LIN {X 0,Y 129.168,Z 1032.646,A -85,B 0,C 180,E1 7073.413,E2 7073.413} C_VEL
LIN {X 0,Y 137.523,Z 1024.267,A -85,B 0,C 180,E1 7063.963,E2 7063.963} C_VEL
LIN {X 0,Y 148.39,Z 1014.459,A -85,B 0,C 180,E1 7056.043,E2 7056.043} C_VEL
LIN {X 0,Y 160.932,Z 1003.211,A -85,B 0,C 180,E1 7049.563,E2 7049.563} C_VEL
LIN {X 0,Y 174.466,Z 990.679,A -85,B 0,C 180,E1 7044.323,E2 7044.323} C_VEL
LIN {X 0,Y 188.456,Z 977.034,A -85,B 0,C 180,E1 7040.101,E2 7040.101} C_VEL
LIN {X 0,Y 202.822,Z 961.714,A -85,B 0,C 180,E1 7036.613,E2 7036.613} C_VEL
LIN {X 0,Y 217.2,Z 944.88,A -85,B 0,C 180,E1 7033.754,E2 7033.754} C_VEL
LIN {X 0,Y 230.71,Z 927.31,A -85,B 0,C 180,E1 7031.498,E2 7031.498} C_VEL
LIN {X 0,Y 243.023,Z 909.185,A -85,B 0,C 180,E1 7029.742,E2 7029.742} C_VEL
LIN {X 0,Y 254.635,Z 889.694,A -85,B 0,C 180,E1 7028.302,E2 7028.302} C_VEL
LIN {X 0,Y 264.561,Z 870.602,A -85,B 0,C 180,E1 7027.217,E2 7027.217} C_VEL
LIN {X 0,Y 273.322,Z 850.557,A -85,B 0,C 180,E1 7026.358,E2 7026.358} C_VEL
LIN {X 0,Y 281.328,Z 828.424,A -85,B 0,C 180,E1 7025.647,E2 7025.647} C_VEL
LIN {X 0,Y 287.652,Z 806.092,A -85,B 0,C 180,E1 7025.074,E2 7025.074} C_VEL
LIN {X 0,Y 292.242,Z 783.432,A -85,B 0,C 180,E1 7024.59,E2 7024.59} C_VEL
LIN {X 0,Y 296.797,Z 747.071,A -85,B 0,C 180,E1 7023.93,E2 7023.93} C_VEL
LIN {X 0,Y 309.195,Z 637.344,A -85,B 0,C 180,E1 7021.992,E2 7021.992} C_VEL
LIN {X 0,Y 308.31,Z 635.045,A -85,B 0,C 180,E1 7019.999,E2 7019.999} C_VEL
LIN {X 0,Y 307.563,Z 632.464,A -85,B 0,C 180,E1 7017.018,E2 7017.018} C_VEL
LIN {X 0,Y 307.478,Z 632.463,A -85,B 0,C 180,E1 7012.663,E2 7012.663} C_VEL
LIN {X 0,Y 308.466,Z 636.029,A -85,B 0,C 180,E1 7008.785,E2 7008.785} C_VEL
LIN {X 0,Y 308.571,Z 636.609,A -85,B 0,C 180,E1 7008.484,E2 7008.484} C_VEL
LIN {X 0,Y 293.648,Z 770.192,A -85,B 0,C 180,E1 7006.284,E2 7006.284} C_VEL
LIN {X 0,Y 289.742,Z 791.809,A -85,B 0,C 180,E1 7005.734,E2 7005.734} C_VEL
LIN {X 0,Y 284.597,Z 812.246,A -85,B 0,C 180,E1 7005.05,E2 7005.05} C_VEL
LIN {X 0,Y 277.983,Z 832.312,A -85,B 0,C 180,E1 7004.188,E2 7004.188} C_VEL
LIN {X 0,Y 270.077,Z 851.641,A -85,B 0,C 180,E1 7003.139,E2 7003.139} C_VEL
LIN {X 0,Y 260.928,Z 870.394,A -85,B 0,C 180,E1 7001.866,E2 7001.866} C_VEL
LIN {X 0,Y 250.585,Z 888.261,A -85,B 0,C 180,E1 7000.334,E2 7000.334} C_VEL
LIN {X 0,Y 239.316,Z 905.023,A -85,B 0,C 180,E1 6998.52,E2 6998.52} C_VEL
LIN {X 0,Y 227.072,Z 920.973,A -85,B 0,C 180,E1 6996.332,E2 6996.332} C_VEL
LIN {X 0,Y 214.134,Z 935.705,A -85,B 0,C 180,E1 6993.704,E2 6993.704} C_VEL
LIN {X 0,Y 200.856,Z 949.005,A -85,B 0,C 180,E1 6990.593,E2 6990.593} C_VEL
LIN {X 0,Y 187.475,Z 961.017,A -85,B 0,C 180,E1 6986.86,E2 6986.86} C_VEL
LIN {X 0,Y 174.234,Z 971.657,A -85,B 0,C 180,E1 6982.367,E2 6982.367} C_VEL
LIN {X 0,Y 161.499,Z 980.804,A -85,B 0,C 180,E1 6976.933,E2 6976.933} C_VEL
LIN {X 0,Y 149.251,Z 988.867,A -85,B 0,C 180,E1 6970.025,E2 6970.025} C_VEL
LIN {X 0,Y 139.655,Z 994.788,A -85,B 0,C 180,E1 6962.477,E2 6962.477} C_VEL
LIN {X 0,Y 132.062,Z 999.229,A -85,B 0,C 180,E1 6953.634,E2 6953.634} C_VEL
LIN {X 0,Y 127.304,Z 1001.968,A -85,B 0,C 180,E1 6944.092,E2 6944.092} C_VEL
LIN {X 0,Y 125.173,Z 1003.266,A -85,B 0,C 180,E1 6934.123,E2 6934.123} C_VEL
LIN {X 0,Y 125.206,Z 1003.258,A -85,B 0,C 180,E1 6925.42,E2 6925.42} C_VEL
LIN {X 0,Y 127.437,Z 1001.916,A -85,B 0,C 180,E1 6915.459,E2 6915.459} C_VEL
LIN {X 0,Y 132.311,Z 999.12,A -85,B 0,C 180,E1 6905.916,E2 6905.916} C_VEL
LIN {X 0,Y 140,Z 994.662,A -85,B 0,C 180,E1 6897.127,E2 6897.127} C_VEL
LIN {X 0,Y 149.777,Z 988.636,A -85,B 0,C 180,E1 6889.556,E2 6889.556} C_VEL
LIN {X 0,Y 162.013,Z 980.566,A -85,B 0,C 180,E1 6882.743,E2 6882.743} C_VEL
LIN {X 0,Y 174.948,Z 971.227,A -85,B 0,C 180,E1 6877.288,E2 6877.288} C_VEL
LIN {X 0,Y 188.83,Z 960.069,A -85,B 0,C 180,E1 6872.657,E2 6872.657} C_VEL
LIN {X 0,Y 202.291,Z 947.848,A -85,B 0,C 180,E1 6868.971,E2 6868.971} C_VEL
LIN {X 0,Y 216.428,Z 933.414,A -85,B 0,C 180,E1 6865.727,E2 6865.727} C_VEL
LIN {X 0,Y 229.449,Z 918.328,A -85,B 0,C 180,E1 6863.151,E2 6863.151} C_VEL
LIN {X 0,Y 241.141,Z 902.814,A -85,B 0,C 180,E1 6861.102,E2 6861.102} C_VEL
LIN {X 0,Y 252.636,Z 885.258,A -85,B 0,C 180,E1 6859.279,E2 6859.279} C_VEL
LIN {X 0,Y 263.01,Z 866.832,A -85,B 0,C 180,E1 6857.767,E2 6857.767} C_VEL
LIN {X 0,Y 272.187,Z 847.478,A -85,B 0,C 180,E1 6856.51,E2 6856.51} C_VEL
LIN {X 0,Y 279.844,Z 827.707,A -85,B 0,C 180,E1 6855.495,E2 6855.495} C_VEL
LIN {X 0,Y 286.583,Z 805.859,A -85,B 0,C 180,E1 6854.618,E2 6854.618} C_VEL
LIN {X 0,Y 291.486,Z 784.725,A -85,B 0,C 180,E1 6853.967,E2 6853.967} C_VEL
LIN {X 0,Y 294.809,Z 763.059,A -85,B 0,C 180,E1 6853.473,E2 6853.473} C_VEL
LIN {X 0,Y 308.856,Z 636.573,A -85,B 0,C 180,E1 6851.39,E2 6851.39} C_VEL
LIN {X 0,Y 308.132,Z 634.469,A -85,B 0,C 180,E1 6849.338,E2 6849.338} C_VEL
LIN {X 0,Y 307.66,Z 632.494,A -85,B 0,C 180,E1 6846.719,E2 6846.719} C_VEL
LIN {X 0,Y 307.835,Z 632.739,A -85,B 0,C 180,E1 6842.793,E2 6842.793} C_VEL
LIN {X 0,Y 309.082,Z 636.612,A -85,B 0,C 180,E1 6838.703,E2 6838.703} C_VEL
LIN {X 0,Y 309.408,Z 637.777,A -85,B 0,C 180,E1 6837.963,E2 6837.963} C_VEL
LIN {X 0,Y 296.291,Z 753.366,A -85,B 0,C 180,E1 6835.967,E2 6835.967} C_VEL
LIN {X 0,Y 295.27,Z 761.06,A -85,B 0,C 180,E1 6836.032,E2 6836.032} C_VEL
LIN {X 0,Y 291.656,Z 781.543,A -85,B 0,C 180,E1 6836.883,E2 6836.883} C_VEL
LIN {X 0,Y 290.371,Z 788.084,A -85,B 0,C 180,E1 6836.883,E2 6836.883} C_VEL
LIN {X 0,Y 284.988,Z 811.855,A -85,B 0,C 180,E1 6836.38,E2 6836.38} C_VEL
LIN {X 0,Y 278.446,Z 833.355,A -85,B 0,C 180,E1 6835.84,E2 6835.84} C_VEL
LIN {X 0,Y 269.935,Z 855.2,A -85,B 0,C 180,E1 6835.14,E2 6835.14} C_VEL
LIN {X 0,Y 260.279,Z 875.739,A -85,B 0,C 180,E1 6834.24,E2 6834.24} C_VEL
LIN {X 0,Y 249.372,Z 895.581,A -85,B 0,C 180,E1 6833.092,E2 6833.092} C_VEL
LIN {X 0,Y 237.943,Z 913.511,A -85,B 0,C 180,E1 6831.73,E2 6831.73} C_VEL
LIN {X 0,Y 224.47,Z 932.114,A -85,B 0,C 180,E1 6829.87,E2 6829.87} C_VEL
LIN {X 0,Y 210.848,Z 948.889,A -85,B 0,C 180,E1 6827.654,E2 6827.654} C_VEL
LIN {X 0,Y 196.469,Z 964.671,A -85,B 0,C 180,E1 6824.862,E2 6824.862} C_VEL
LIN {X 0,Y 181.547,Z 979.576,A -85,B 0,C 180,E1 6821.314,E2 6821.314} C_VEL
LIN {X 0,Y 166.472,Z 993.481,A -85,B 0,C 180,E1 6816.773,E2 6816.773} C_VEL
LIN {X 0,Y 151.986,Z 1005.938,A -85,B 0,C 180,E1 6811.04,E2 6811.04} C_VEL
LIN {X 0,Y 138.719,Z 1016.968,A -85,B 0,C 180,E1 6803.831,E2 6803.831} C_VEL
LIN {X 0,Y 127.52,Z 1026.514,A -85,B 0,C 180,E1 6794.884,E2 6794.884} C_VEL
LIN {X 0,Y 119.945,Z 1033.8,A -85,B 0,C 180,E1 6785.113,E2 6785.113} C_VEL
LIN {X 0,Y 115.716,Z 1039.287,A -85,B 0,C 180,E1 6774.504,E2 6774.504} C_VEL
LIN {X 0,Y 114.694,Z 1042.845,A -85,B 0,C 180,E1 6764.619,E2 6764.619} C_VEL
LIN {X 0,Y 115.455,Z 1044.705,A -85,B 0,C 180,E1 6755.965,E2 6755.965} C_VEL
LIN {X 0,Y 116.042,Z 1045.172,A -85,B 0,C 180,E1 6750.494,E2 6750.494} C_VEL
LIN {X 0,Y 115.673,Z 1044.857,A -85,B 0,C 180,E1 6745.538,E2 6745.538} C_VEL
LIN {X 0,Y 114.765,Z 1043.356,A -85,B 0,C 180,E1 6737.354,E2 6737.354} C_VEL
LIN {X 0,Y 115.389,Z 1039.917,A -85,B 0,C 180,E1 6727.05,E2 6727.05} C_VEL
LIN {X 0,Y 118.623,Z 1035.213,A -85,B 0,C 180,E1 6717.354,E2 6717.354} C_VEL
LIN {X 0,Y 125.827,Z 1027.96,A -85,B 0,C 180,E1 6706.891,E2 6706.891} C_VEL
LIN {X 0,Y 135.903,Z 1019.293,A -85,B 0,C 180,E1 6698.073,E2 6698.073} C_VEL
LIN {X 0,Y 147.961,Z 1009.202,A -85,B 0,C 180,E1 6690.882,E2 6690.882} C_VEL
LIN {X 0,Y 162.033,Z 997.214,A -85,B 0,C 180,E1 6684.809,E2 6684.809} C_VEL
LIN {X 0,Y 176.659,Z 984.102,A -85,B 0,C 180,E1 6680.026,E2 6680.026} C_VEL
LIN {X 0,Y 191.59,Z 969.538,A -85,B 0,C 180,E1 6676.207,E2 6676.207} C_VEL
LIN {X 0,Y 206.378,Z 953.698,A -85,B 0,C 180,E1 6673.142,E2 6673.142} C_VEL
LIN {X 0,Y 220.798,Z 936.614,A -85,B 0,C 180,E1 6670.683,E2 6670.683} C_VEL
LIN {X 0,Y 233.725,Z 919.31,A -85,B 0,C 180,E1 6668.807,E2 6668.807} C_VEL
LIN {X 0,Y 245.951,Z 900.785,A -85,B 0,C 180,E1 6667.282,E2 6667.282} C_VEL
LIN {X 0,Y 256.915,Z 881.888,A -85,B 0,C 180,E1 6666.087,E2 6666.087} C_VEL
LIN {X 0,Y 267.025,Z 861.28,A -85,B 0,C 180,E1 6665.106,E2 6665.106} C_VEL
LIN {X 0,Y 276.006,Z 839.357,A -85,B 0,C 180,E1 6664.342,E2 6664.342} C_VEL
LIN {X 0,Y 283.32,Z 817.128,A -85,B 0,C 180,E1 6663.751,E2 6663.751} C_VEL
LIN {X 0,Y 288.927,Z 794.538,A -85,B 0,C 180,E1 6663.252,E2 6663.252} C_VEL
LIN {X 0,Y 292.707,Z 771.832,A -85,B 0,C 180,E1 6662.822,E2 6662.822} C_VEL
LIN {X 0,Y 307.568,Z 643.681,A -85,B 0,C 180,E1 6660.651,E2 6660.651} C_VEL
LIN {X 0,Y 306.554,Z 640.371,A -85,B 0,C 180,E1 6656.821,E2 6656.821} C_VEL
LIN {X 0,Y 306.492,Z 640.482,A -85,B 0,C 180,E1 6652.69,E2 6652.69} C_VEL
LIN {X 0,Y 307.068,Z 643.011,A -85,B 0,C 180,E1 6649.87,E2 6649.87} C_VEL
LIN {X 0,Y 292.446,Z 770.849,A -85,B 0,C 180,E1 6647.825,E2 6647.825} C_VEL
LIN {X 0,Y 288.464,Z 792.458,A -85,B 0,C 180,E1 6647.294,E2 6647.294} C_VEL
LIN {X 0,Y 283.142,Z 813.196,A -85,B 0,C 180,E1 6646.626,E2 6646.626} C_VEL
LIN {X 0,Y 276.411,Z 833.238,A -85,B 0,C 180,E1 6645.799,E2 6645.799} C_VEL
LIN {X 0,Y 268.363,Z 852.557,A -85,B 0,C 180,E1 6644.793,E2 6644.793} C_VEL
LIN {X 0,Y 259.043,Z 871.321,A -85,B 0,C 180,E1 6643.572,E2 6643.572} C_VEL
LIN {X 0,Y 248.495,Z 889.202,A -85,B 0,C 180,E1 6642.102,E2 6642.102} C_VEL
LIN {X 0,Y 236.791,Z 906.255,A -85,B 0,C 180,E1 6640.328,E2 6640.328} C_VEL
LIN {X 0,Y 224.876,Z 921.49,A -85,B 0,C 180,E1 6638.323,E2 6638.323} C_VEL
LIN {X 0,Y 211.579,Z 936.29,A -85,B 0,C 180,E1 6635.792,E2 6635.792} C_VEL
LIN {X 0,Y 197.89,Z 949.707,A -85,B 0,C 180,E1 6632.781,E2 6632.781} C_VEL
LIN {X 0,Y 184.024,Z 961.824,A -85,B 0,C 180,E1 6629.145,E2 6629.145} C_VEL
LIN {X 0,Y 170.215,Z 972.521,A -85,B 0,C 180,E1 6624.736,E2 6624.736} C_VEL
LIN {X 0,Y 156.826,Z 981.768,A -85,B 0,C 180,E1 6619.35,E2 6619.35} C_VEL
LIN {X 0,Y 144.365,Z 989.606,A -85,B 0,C 180,E1 6612.746,E2 6612.746} C_VEL
LIN {X 0,Y 133.912,Z 995.704,A -85,B 0,C 180,E1 6605.095,E2 6605.095} C_VEL
LIN {X 0,Y 125.479,Z 1000.232,A -85,B 0,C 180,E1 6595.993,E2 6595.993} C_VEL
LIN {X 0,Y 120.003,Z 1003.146,A -85,B 0,C 180,E1 6585.959,E2 6585.959} C_VEL
LIN {X 0,Y 117.473,Z 1004.583,A -85,B 0,C 180,E1 6575.862,E2 6575.862} C_VEL
LIN {X 0,Y 117.248,Z 1004.661,A -85,B 0,C 180,E1 6566.174,E2 6566.174} C_VEL
LIN {X 0,Y 119.465,Z 1003.476,A -85,B 0,C 180,E1 6555.458,E2 6555.458} C_VEL
LIN {X 0,Y 124.517,Z 1000.849,A -85,B 0,C 180,E1 6545.319,E2 6545.319} C_VEL
LIN {X 0,Y 132.538,Z 996.484,A -85,B 0,C 180,E1 6536.065,E2 6536.065} C_VEL
LIN {X 0,Y 143.196,Z 990.387,A -85,B 0,C 180,E1 6527.908,E2 6527.908} C_VEL
LIN {X 0,Y 156.111,Z 982.368,A -85,B 0,C 180,E1 6520.907,E2 6520.907} C_VEL
LIN {X 0,Y 169.428,Z 973.26,A -85,B 0,C 180,E1 6515.472,E2 6515.472} C_VEL
LIN {X 0,Y 183.179,Z 962.654,A -85,B 0,C 180,E1 6511.022,E2 6511.022} C_VEL
LIN {X 0,Y 197.009,Z 950.72,A -85,B 0,C 180,E1 6507.356,E2 6507.356} C_VEL
LIN {X 0,Y 210.672,Z 937.502,A -85,B 0,C 180,E1 6504.322,E2 6504.322} C_VEL
LIN {X 0,Y 224.136,Z 922.594,A -85,B 0,C 180,E1 6501.732,E2 6501.732} C_VEL
LIN {X 0,Y 236.704,Z 906.685,A -85,B 0,C 180,E1 6499.613,E2 6499.613} C_VEL
LIN {X 0,Y 248.412,Z 889.718,A -85,B 0,C 180,E1 6497.839,E2 6497.839} C_VEL
LIN {X 0,Y 258.896,Z 871.998,A -85,B 0,C 180,E1 6496.376,E2 6496.376} C_VEL
LIN {X 0,Y 268.285,Z 853.243,A -85,B 0,C 180,E1 6495.146,E2 6495.146} C_VEL
LIN {X 0,Y 276.339,Z 834.11,A -85,B 0,C 180,E1 6494.142,E2 6494.142} C_VEL
LIN {X 0,Y 283.07,Z 814.201,A -85,B 0,C 180,E1 6493.313,E2 6493.313} C_VEL
LIN {X 0,Y 288.641,Z 792.794,A -85,B 0,C 180,E1 6492.619,E2 6492.619} C_VEL
LIN {X 0,Y 292.691,Z 770.866,A -85,B 0,C 180,E1 6492.078,E2 6492.078} C_VEL
LIN {X 0,Y 307.388,Z 643.047,A -85,B 0,C 180,E1 6490.032,E2 6490.032} C_VEL
LIN {X 0,Y 306.668,Z 640.418,A -85,B 0,C 180,E1 6486.553,E2 6486.553} C_VEL
LIN {X 0,Y 306.827,Z 640.61,A -85,B 0,C 180,E1 6482.989,E2 6482.989} C_VEL
LIN {X 0,Y 307.792,Z 643.979,A -85,B 0,C 180,E1 6479.341,E2 6479.341} C_VEL
LIN {X 0,Y 291.953,Z 779.066,A -85,B 0,C 180,E1 6477.056,E2 6477.056} C_VEL
LIN {X 0,Y 290.371,Z 788.084,A -85,B 0,C 180,E1 6476.883,E2 6476.883} C_VEL
LIN {X 0,Y 288.487,Z 796.75,A -85,B 0,C 180,E1 6476.959,E2 6476.959} C_VEL
LIN {X 0,Y 283.247,Z 814.649,A -85,B 0,C 180,E1 6477.719,E2 6477.719} C_VEL
LIN {X 0,Y 280.857,Z 822.038,A -85,B 0,C 180,E1 6477.749,E2 6477.749} C_VEL
LIN {X 0,Y 273.293,Z 843.641,A -85,B 0,C 180,E1 6477.187,E2 6477.187} C_VEL
LIN {X 0,Y 264.46,Z 863.924,A -85,B 0,C 180,E1 6476.495,E2 6476.495} C_VEL
LIN {X 0,Y 253.739,Z 884.733,A -85,B 0,C 180,E1 6475.528,E2 6475.528} C_VEL
LIN {X 0,Y 241.855,Z 904.472,A -85,B 0,C 180,E1 6474.307,E2 6474.307} C_VEL
LIN {X 0,Y 228.794,Z 923.101,A -85,B 0,C 180,E1 6472.76,E2 6472.76} C_VEL
LIN {X 0,Y 214.271,Z 941.356,A -85,B 0,C 180,E1 6470.729,E2 6470.729} C_VEL
LIN {X 0,Y 199.18,Z 958.205,A -85,B 0,C 180,E1 6468.204,E2 6468.204} C_VEL
LIN {X 0,Y 184.148,Z 973.242,A -85,B 0,C 180,E1 6465.125,E2 6465.125} C_VEL
LIN {X 0,Y 168.946,Z 987.038,A -85,B 0,C 180,E1 6461.249,E2 6461.249} C_VEL
LIN {X 0,Y 153.586,Z 999.968,A -85,B 0,C 180,E1 6456.196,E2 6456.196} C_VEL
LIN {X 0,Y 138.967,Z 1011.527,A -85,B 0,C 180,E1 6449.701,E2 6449.701} C_VEL
LIN {X 0,Y 126.225,Z 1021.348,A -85,B 0,C 180,E1 6441.647,E2 6441.647} C_VEL
LIN {X 0,Y 115.942,Z 1029.738,A -85,B 0,C 180,E1 6431.608,E2 6431.608} C_VEL
LIN {X 0,Y 109.765,Z 1035.768,A -85,B 0,C 180,E1 6421.105,E2 6421.105} C_VEL
LIN {X 0,Y 106.923,Z 1040.415,A -85,B 0,C 180,E1 6409.105,E2 6409.105} C_VEL
LIN {X 0,Y 107.097,Z 1042.759,A -85,B 0,C 180,E1 6399.674,E2 6399.674} C_VEL
LIN {X 0,Y 108.056,Z 1043.707,A -85,B 0,C 180,E1 6392.121,E2 6392.121} C_VEL
LIN {X 0,Y 108.056,Z 1043.702,A -85,B 0,C 180,E1 6387.865,E2 6387.865} C_VEL
LIN {X 0,Y 107.097,Z 1042.746,A -85,B 0,C 180,E1 6380.325,E2 6380.325} C_VEL
LIN {X 0,Y 106.935,Z 1040.364,A -85,B 0,C 180,E1 6370.792,E2 6370.792} C_VEL
LIN {X 0,Y 109.83,Z 1035.655,A -85,B 0,C 180,E1 6358.74,E2 6358.74} C_VEL
LIN {X 0,Y 115.94,Z 1029.692,A -85,B 0,C 180,E1 6348.391,E2 6348.391} C_VEL
LIN {X 0,Y 125.683,Z 1021.706,A -85,B 0,C 180,E1 6338.772,E2 6338.772} C_VEL
LIN {X 0,Y 138.303,Z 1011.975,A -85,B 0,C 180,E1 6330.648,E2 6330.648} C_VEL
LIN {X 0,Y 152.423,Z 1000.778,A -85,B 0,C 180,E1 6324.242,E2 6324.242} C_VEL
LIN {X 0,Y 168.123,Z 987.622,A -85,B 0,C 180,E1 6318.984,E2 6318.984} C_VEL
LIN {X 0,Y 183.278,Z 973.924,A -85,B 0,C 180,E1 6315.068,E2 6315.068} C_VEL
LIN {X 0,Y 198.482,Z 958.727,A -85,B 0,C 180,E1 6311.919,E2 6311.919} C_VEL
LIN {X 0,Y 213.017,Z 942.589,A -85,B 0,C 180,E1 6309.455,E2 6309.455} C_VEL
LIN {X 0,Y 226.899,Z 925.402,A -85,B 0,C 180,E1 6307.476,E2 6307.476} C_VEL
LIN {X 0,Y 239.746,Z 907.253,A -85,B 0,C 180,E1 6305.917,E2 6305.917} C_VEL
LIN {X 0,Y 251.796,Z 887.736,A -85,B 0,C 180,E1 6304.651,E2 6304.651} C_VEL
LIN {X 0,Y 262.503,Z 867.622,A -85,B 0,C 180,E1 6303.668,E2 6303.668} C_VEL
LIN {X 0,Y 271.325,Z 847.873,A -85,B 0,C 180,E1 6302.955,E2 6302.955} C_VEL
LIN {X 0,Y 279.201,Z 826.422,A -85,B 0,C 180,E1 6302.366,E2 6302.366} C_VEL
LIN {X 0,Y 285.552,Z 804.428,A -85,B 0,C 180,E1 6301.871,E2 6301.871} C_VEL
LIN {X 0,Y 290.209,Z 781.99,A -85,B 0,C 180,E1 6301.439,E2 6301.439} C_VEL
LIN {X 0,Y 294.604,Z 748.025,A -85,B 0,C 180,E1 6300.864,E2 6300.864} C_VEL
LIN {X 0,Y 306.041,Z 650.45,A -85,B 0,C 180,E1 6299.251,E2 6299.251} C_VEL
LIN {X 0,Y 305.538,Z 648.282,A -85,B 0,C 180,E1 6296.623,E2 6296.623} C_VEL
LIN {X 0,Y 305.497,Z 648.381,A -85,B 0,C 180,E1 6292.855,E2 6292.855} C_VEL
LIN {X 0,Y 305.695,Z 649.877,A -85,B 0,C 180,E1 6291.262,E2 6291.262} C_VEL
LIN {X 0,Y 291.442,Z 771.609,A -85,B 0,C 180,E1 6289.376,E2 6289.376} C_VEL
LIN {X 0,Y 287.374,Z 793.238,A -85,B 0,C 180,E1 6288.864,E2 6288.864} C_VEL
LIN {X 0,Y 281.903,Z 814.147,A -85,B 0,C 180,E1 6288.217,E2 6288.217} C_VEL
LIN {X 0,Y 275.157,Z 833.898,A -85,B 0,C 180,E1 6287.439,E2 6287.439} C_VEL
LIN {X 0,Y 266.876,Z 853.472,A -85,B 0,C 180,E1 6286.466,E2 6286.466} C_VEL
LIN {X 0,Y 257.391,Z 872.246,A -85,B 0,C 180,E1 6285.301,E2 6285.301} C_VEL
LIN {X 0,Y 246.645,Z 890.141,A -85,B 0,C 180,E1 6283.897,E2 6283.897} C_VEL
LIN {X 0,Y 234.705,Z 907.222,A -85,B 0,C 180,E1 6282.201,E2 6282.201} C_VEL
LIN {X 0,Y 222.091,Z 922.974,A -85,B 0,C 180,E1 6280.208,E2 6280.208} C_VEL
LIN {X 0,Y 208.474,Z 937.753,A -85,B 0,C 180,E1 6277.767,E2 6277.767} C_VEL
LIN {X 0,Y 194.408,Z 951.135,A -85,B 0,C 180,E1 6274.849,E2 6274.849} C_VEL
LIN {X 0,Y 180.098,Z 963.223,A -85,B 0,C 180,E1 6271.305,E2 6271.305} C_VEL
LIN {X 0,Y 165.774,Z 973.918,A -85,B 0,C 180,E1 6266.97,E2 6266.97} C_VEL
LIN {X 0,Y 151.784,Z 983.155,A -85,B 0,C 180,E1 6261.62,E2 6261.62} C_VEL
LIN {X 0,Y 138.065,Z 991.298,A -85,B 0,C 180,E1 6254.626,E2 6254.626} C_VEL
LIN {X 0,Y 127.029,Z 997.31,A -85,B 0,C 180,E1 6246.742,E2 6246.742} C_VEL
LIN {X 0,Y 118.069,Z 1001.787,A -85,B 0,C 180,E1 6237.213,E2 6237.213} C_VEL
LIN {X 0,Y 112.224,Z 1004.609,A -85,B 0,C 180,E1 6226.565,E2 6226.565} C_VEL
LIN {X 0,Y 109.562,Z 1005.964,A -85,B 0,C 180,E1 6215.762,E2 6215.762} C_VEL
LIN {X 0,Y 109.388,Z 1006.024,A -85,B 0,C 180,E1 6205.807,E2 6205.807} C_VEL
LIN {X 0,Y 111.832,Z 1004.845,A -85,B 0,C 180,E1 6194.441,E2 6194.441} C_VEL
LIN {X 0,Y 117.364,Z 1002.22,A -85,B 0,C 180,E1 6183.704,E2 6183.704} C_VEL
LIN {X 0,Y 126.156,Z 997.795,A -85,B 0,C 180,E1 6173.943,E2 6173.943} C_VEL
LIN {X 0,Y 137.413,Z 991.761,A -85,B 0,C 180,E1 6165.691,E2 6165.691} C_VEL
LIN {X 0,Y 150.381,Z 984.171,A -85,B 0,C 180,E1 6158.929,E2 6158.929} C_VEL
LIN {X 0,Y 164.233,Z 975.143,A -85,B 0,C 180,E1 6153.481,E2 6153.481} C_VEL
LIN {X 0,Y 178.458,Z 964.644,A -85,B 0,C 180,E1 6149.069,E2 6149.069} C_VEL
LIN {X 0,Y 193.509,Z 952.138,A -85,B 0,C 180,E1 6145.28,E2 6145.28} C_VEL
LIN {X 0,Y 207.552,Z 938.958,A -85,B 0,C 180,E1 6142.34,E2 6142.34} C_VEL
LIN {X 0,Y 221.143,Z 924.293,A -85,B 0,C 180,E1 6139.874,E2 6139.874} C_VEL
LIN {X 0,Y 234.185,Z 908.224,A -85,B 0,C 180,E1 6137.804,E2 6137.804} C_VEL
LIN {X 0,Y 246.126,Z 891.355,A -85,B 0,C 180,E1 6136.103,E2 6136.103} C_VEL
LIN {X 0,Y 256.866,Z 873.582,A -85,B 0,C 180,E1 6134.692,E2 6134.692} C_VEL
LIN {X 0,Y 266.806,Z 854.148,A -85,B 0,C 180,E1 6133.471,E2 6133.471} C_VEL
LIN {X 0,Y 274.996,Z 835.02,A -85,B 0,C 180,E1 6132.513,E2 6132.513} C_VEL
LIN {X 0,Y 281.839,Z 815.133,A -85,B 0,C 180,E1 6131.721,E2 6131.721} C_VEL
LIN {X 0,Y 287.554,Z 793.588,A -85,B 0,C 180,E1 6131.05,E2 6131.05} C_VEL
LIN {X 0,Y 291.686,Z 771.686,A -85,B 0,C 180,E1 6130.53,E2 6130.53} C_VEL
LIN {X 0,Y 305.99,Z 649.959,A -85,B 0,C 180,E1 6128.645,E2 6128.645} C_VEL
LIN {X 0,Y 305.681,Z 648.342,A -85,B 0,C 180,E1 6126.386,E2 6126.386} C_VEL
LIN {X 0,Y 305.841,Z 648.653,A -85,B 0,C 180,E1 6122.999,E2 6122.999} C_VEL
LIN {X 0,Y 306.268,Z 650.919,A -85,B 0,C 180,E1 6120.721,E2 6120.721} C_VEL
LIN {X 0,Y 291.044,Z 778.478,A -85,B 0,C 180,E1 6118.631,E2 6118.631} C_VEL
LIN {X 0,Y 286.602,Z 800.907,A -85,B 0,C 180,E1 6118.206,E2 6118.206} C_VEL
LIN {X 0,Y 280.857,Z 822.038,A -85,B 0,C 180,E1 6117.749,E2 6117.749} C_VEL
LIN {X 0,Y 278.71,Z 828.32,A -85,B 0,C 180,E1 6117.788,E2 6117.788} C_VEL
LIN {X 0,Y 271.025,Z 846.672,A -85,B 0,C 180,E1 6118.528,E2 6118.528} C_VEL
LIN {X 0,Y 267.887,Z 853.694,A -85,B 0,C 180,E1 6118.555,E2 6118.555} C_VEL
LIN {X 0,Y 267.456,Z 854.699,A -85,B 0,C 180,E1 6118.529,E2 6118.529} C_VEL
LIN {X 0,Y 257.707,Z 874.676,A -85,B 0,C 180,E1 6117.777,E2 6117.777} C_VEL
LIN {X 0,Y 246.356,Z 894.548,A -85,B 0,C 180,E1 6116.779,E2 6116.779} C_VEL
LIN {X 0,Y 234.221,Z 912.856,A -85,B 0,C 180,E1 6115.562,E2 6115.562} C_VEL
LIN {X 0,Y 221.038,Z 930.208,A -85,B 0,C 180,E1 6114.029,E2 6114.029} C_VEL
LIN {X 0,Y 206.003,Z 947.754,A -85,B 0,C 180,E1 6111.949,E2 6111.949} C_VEL
LIN {X 0,Y 190.924,Z 963.362,A -85,B 0,C 180,E1 6109.439,E2 6109.439} C_VEL
LIN {X 0,Y 174.687,Z 978.393,A -85,B 0,C 180,E1 6106.091,E2 6106.091} C_VEL
LIN {X 0,Y 157.987,Z 992.406,A -85,B 0,C 180,E1 6101.681,E2 6101.681} C_VEL
LIN {X 0,Y 142.161,Z 1004.676,A -85,B 0,C 180,E1 6096.112,E2 6096.112} C_VEL
LIN {X 0,Y 127.337,Z 1015.413,A -85,B 0,C 180,E1 6088.857,E2 6088.857} C_VEL
LIN {X 0,Y 114.46,Z 1024.672,A -85,B 0,C 180,E1 6079.463,E2 6079.463} C_VEL
LIN {X 0,Y 105.447,Z 1031.771,A -85,B 0,C 180,E1 6068.743,E2 6068.743} C_VEL
LIN {X 0,Y 100.221,Z 1037.052,A -85,B 0,C 180,E1 6056.676,E2 6056.676} C_VEL
LIN {X 0,Y 98.852,Z 1040.548,A -85,B 0,C 180,E1 6044.647,E2 6044.647} C_VEL
LIN {X 0,Y 99.737,Z 1042.092,A -85,B 0,C 180,E1 6035.176,E2 6035.176} C_VEL
LIN {X 0,Y 100.286,Z 1042.459,A -85,B 0,C 180,E1 6030,E2 6030} C_VEL
LIN {X 0,Y 99.649,Z 1042.032,A -85,B 0,C 180,E1 6024.241,E2 6024.241} C_VEL
LIN {X 0,Y 98.845,Z 1040.293,A -85,B 0,C 180,E1 6014.15,E2 6014.15} C_VEL
LIN {X 0,Y 100.557,Z 1036.581,A -85,B 0,C 180,E1 6002.138,E2 6002.138} C_VEL
LIN {X 0,Y 106.149,Z 1031.133,A -85,B 0,C 180,E1 5990.169,E2 5990.169} C_VEL
LIN {X 0,Y 115.494,Z 1023.865,A -85,B 0,C 180,E1 5979.601,E2 5979.601} C_VEL
LIN {X 0,Y 128.651,Z 1014.37,A -85,B 0,C 180,E1 5970.381,E2 5970.381} C_VEL
LIN {X 0,Y 143.239,Z 1003.742,A -85,B 0,C 180,E1 5963.444,E2 5963.444} C_VEL
LIN {X 0,Y 158.811,Z 991.641,A -85,B 0,C 180,E1 5958.068,E2 5958.068} C_VEL
LIN {X 0,Y 175.044,Z 977.914,A -85,B 0,C 180,E1 5953.819,E2 5953.819} C_VEL
LIN {X 0,Y 191.18,Z 962.907,A -85,B 0,C 180,E1 5950.506,E2 5950.506} C_VEL
LIN {X 0,Y 206.469,Z 947.04,A -85,B 0,C 180,E1 5947.973,E2 5947.973} C_VEL
LIN {X 0,Y 221.161,Z 929.783,A -85,B 0,C 180,E1 5945.946,E2 5945.946} C_VEL
LIN {X 0,Y 235.139,Z 911.188,A -85,B 0,C 180,E1 5944.328,E2 5944.328} C_VEL
LIN {X 0,Y 247.334,Z 892.642,A -85,B 0,C 180,E1 5943.12,E2 5943.12} C_VEL
LIN {X 0,Y 258.152,Z 873.387,A -85,B 0,C 180,E1 5942.177,E2 5942.177} C_VEL
LIN {X 0,Y 268.047,Z 852.747,A -85,B 0,C 180,E1 5941.42,E2 5941.42} C_VEL
LIN {X 0,Y 276.543,Z 831.321,A -85,B 0,C 180,E1 5940.842,E2 5940.842} C_VEL
LIN {X 0,Y 283.406,Z 809.033,A -85,B 0,C 180,E1 5940.361,E2 5940.361} C_VEL
LIN {X 0,Y 288.65,Z 785.987,A -85,B 0,C 180,E1 5939.931,E2 5939.931} C_VEL
LIN {X 0,Y 292.268,Z 761.823,A -85,B 0,C 180,E1 5939.528,E2 5939.528} C_VEL
LIN {X 0,Y 304.702,Z 657.198,A -85,B 0,C 180,E1 5937.837,E2 5937.837} C_VEL
LIN {X 0,Y 304.518,Z 656.195,A -85,B 0,C 180,E1 5936.423,E2 5936.423} C_VEL
LIN {X 0,Y 304.505,Z 656.279,A -85,B 0,C 180,E1 5933.021,E2 5933.021} C_VEL
LIN {X 0,Y 304.509,Z 656.722,A -85,B 0,C 180,E1 5932.666,E2 5932.666} C_VEL
LIN {X 0,Y 290.654,Z 772.37,A -85,B 0,C 180,E1 5930.936,E2 5930.936} C_VEL
LIN {X 0,Y 286.501,Z 794.03,A -85,B 0,C 180,E1 5930.444,E2 5930.444} C_VEL
LIN {X 0,Y 280.884,Z 815.098,A -85,B 0,C 180,E1 5929.822,E2 5929.822} C_VEL
LIN {X 0,Y 273.934,Z 835.089,A -85,B 0,C 180,E1 5929.07,E2 5929.07} C_VEL
LIN {X 0,Y 265.619,Z 854.389,A -85,B 0,C 180,E1 5928.157,E2 5928.157} C_VEL
LIN {X 0,Y 255.977,Z 873.172,A -85,B 0,C 180,E1 5927.051,E2 5927.051} C_VEL
LIN {X 0,Y 245.042,Z 891.08,A -85,B 0,C 180,E1 5925.718,E2 5925.718} C_VEL
LIN {X 0,Y 232.874,Z 908.189,A -85,B 0,C 180,E1 5924.106,E2 5924.106} C_VEL
LIN {X 0,Y 219.553,Z 924.455,A -85,B 0,C 180,E1 5922.14,E2 5922.14} C_VEL
LIN {X 0,Y 205.624,Z 939.215,A -85,B 0,C 180,E1 5919.798,E2 5919.798} C_VEL
LIN {X 0,Y 191.188,Z 952.562,A -85,B 0,C 180,E1 5916.99,E2 5916.99} C_VEL
LIN {X 0,Y 175.637,Z 965.223,A -85,B 0,C 180,E1 5913.351,E2 5913.351} C_VEL
LIN {X 0,Y 160.842,Z 975.849,A -85,B 0,C 180,E1 5909.078,E2 5909.078} C_VEL
LIN {X 0,Y 146.3,Z 984.964,A -85,B 0,C 180,E1 5903.751,E2 5903.751} C_VEL
LIN {X 0,Y 132.54,Z 992.678,A -85,B 0,C 180,E1 5897.034,E2 5897.034} C_VEL
LIN {X 0,Y 120.765,Z 998.683,A -85,B 0,C 180,E1 5888.994,E2 5888.994} C_VEL
LIN {X 0,Y 111.083,Z 1003.161,A -85,B 0,C 180,E1 5879.082,E2 5879.082} C_VEL
LIN {X 0,Y 104.67,Z 1005.979,A -85,B 0,C 180,E1 5867.799,E2 5867.799} C_VEL
LIN {X 0,Y 101.718,Z 1007.33,A -85,B 0,C 180,E1 5856.208,E2 5856.208} C_VEL
LIN {X 0,Y 101.526,Z 1007.389,A -85,B 0,C 180,E1 5845.481,E2 5845.481} C_VEL
LIN {X 0,Y 104.236,Z 1006.215,A -85,B 0,C 180,E1 5833.276,E2 5833.276} C_VEL
LIN {X 0,Y 110.316,Z 1003.592,A -85,B 0,C 180,E1 5821.881,E2 5821.881} C_VEL
LIN {X 0,Y 119.703,Z 999.226,A -85,B 0,C 180,E1 5811.821,E2 5811.821} C_VEL
LIN {X 0,Y 131.855,Z 993.134,A -85,B 0,C 180,E1 5803.283,E2 5803.283} C_VEL
LIN {X 0,Y 145.531,Z 985.552,A -85,B 0,C 180,E1 5796.501,E2 5796.501} C_VEL
LIN {X 0,Y 160.759,Z 976.041,A -85,B 0,C 180,E1 5790.872,E2 5790.872} C_VEL
LIN {X 0,Y 175.553,Z 965.444,A -85,B 0,C 180,E1 5786.594,E2 5786.594} C_VEL
LIN {X 0,Y 191.107,Z 952.827,A -85,B 0,C 180,E1 5782.952,E2 5782.952} C_VEL
LIN {X 0,Y 205.545,Z 939.533,A -85,B 0,C 180,E1 5780.142,E2 5780.142} C_VEL
LIN {X 0,Y 219.83,Z 924.412,A -85,B 0,C 180,E1 5777.743,E2 5777.743} C_VEL
LIN {X 0,Y 232.8,Z 908.596,A -85,B 0,C 180,E1 5775.831,E2 5775.831} C_VEL
LIN {X 0,Y 244.973,Z 891.578,A -85,B 0,C 180,E1 5774.219,E2 5774.219} C_VEL
LIN {X 0,Y 255.911,Z 873.714,A -85,B 0,C 180,E1 5772.885,E2 5772.885} C_VEL
LIN {X 0,Y 265.557,Z 855.052,A -85,B 0,C 180,E1 5771.779,E2 5771.779} C_VEL
LIN {X 0,Y 274.339,Z 834.688,A -85,B 0,C 180,E1 5770.817,E2 5770.817} C_VEL
LIN {X 0,Y 281.294,Z 814.626,A -85,B 0,C 180,E1 5770.068,E2 5770.068} C_VEL
LIN {X 0,Y 286.892,Z 793.467,A -85,B 0,C 180,E1 5769.448,E2 5769.448} C_VEL
LIN {X 0,Y 291.138,Z 770.761,A -85,B 0,C 180,E1 5768.939,E2 5768.939} C_VEL
LIN {X 0,Y 304.771,Z 656.826,A -85,B 0,C 180,E1 5767.22,E2 5767.22} C_VEL
LIN {X 0,Y 304.684,Z 656.252,A -85,B 0,C 180,E1 5766.028,E2 5766.028} C_VEL
LIN {X 0,Y 304.837,Z 656.523,A -85,B 0,C 180,E1 5763.197,E2 5763.197} C_VEL
LIN {X 0,Y 304.946,Z 657.667,A -85,B 0,C 180,E1 5762.117,E2 5762.117} C_VEL
LIN {X 0,Y 290.345,Z 777.98,A -85,B 0,C 180,E1 5760.213,E2 5760.213} C_VEL
LIN {X 0,Y 285.831,Z 800.411,A -85,B 0,C 180,E1 5759.811,E2 5759.811} C_VEL
LIN {X 0,Y 279.481,Z 823.131,A -85,B 0,C 180,E1 5759.35,E2 5759.35} C_VEL
LIN {X 0,Y 272.019,Z 843.967,A -85,B 0,C 180,E1 5758.846,E2 5758.846} C_VEL
LIN {X 0,Y 267.456,Z 854.699,A -85,B 0,C 180,E1 5758.529,E2 5758.529} C_VEL
LIN {X 0,Y 264.152,Z 861.732,A -85,B 0,C 180,E1 5758.513,E2 5758.513} C_VEL
LIN {X 0,Y 254.308,Z 879.08,A -85,B 0,C 180,E1 5759.151,E2 5759.151} C_VEL
LIN {X 0,Y 250.309,Z 885.673,A -85,B 0,C 180,E1 5759.076,E2 5759.076} C_VEL
LIN {X 0,Y 237.647,Z 905.544,A -85,B 0,C 180,E1 5757.988,E2 5757.988} C_VEL
LIN {X 0,Y 224.352,Z 923.655,A -85,B 0,C 180,E1 5756.657,E2 5756.657} C_VEL
LIN {X 0,Y 209.791,Z 940.884,A -85,B 0,C 180,E1 5754.936,E2 5754.936} C_VEL
LIN {X 0,Y 193.168,Z 958.261,A -85,B 0,C 180,E1 5752.566,E2 5752.566} C_VEL
LIN {X 0,Y 176.845,Z 973.441,A -85,B 0,C 180,E1 5749.666,E2 5749.666} C_VEL
LIN {X 0,Y 159.838,Z 987.551,A -85,B 0,C 180,E1 5745.837,E2 5745.837} C_VEL
LIN {X 0,Y 143.741,Z 999.637,A -85,B 0,C 180,E1 5741.089,E2 5741.089} C_VEL
LIN {X 0,Y 127.412,Z 1011.035,A -85,B 0,C 180,E1 5734.484,E2 5734.484} C_VEL
LIN {X 0,Y 113.21,Z 1020.499,A -85,B 0,C 180,E1 5726.12,E2 5726.12} C_VEL
LIN {X 0,Y 101.929,Z 1028.083,A -85,B 0,C 180,E1 5715.733,E2 5715.733} C_VEL
LIN {X 0,Y 94.124,Z 1034.263,A -85,B 0,C 180,E1 5702.804,E2 5702.804} C_VEL
LIN {X 0,Y 91.107,Z 1038.222,A -85,B 0,C 180,E1 5689.89,E2 5689.89} C_VEL
LIN {X 0,Y 91.408,Z 1040.465,A -85,B 0,C 180,E1 5678.175,E2 5678.175} C_VEL
LIN {X 0,Y 92.334,Z 1041.04,A -85,B 0,C 180,E1 5671.241,E2 5671.241} C_VEL
LIN {X 0,Y 92.12,Z 1040.908,A -85,B 0,C 180,E1 5666.879,E2 5666.879} C_VEL
LIN {X 0,Y 91.041,Z 1039.786,A -85,B 0,C 180,E1 5657.798,E2 5657.798} C_VEL
LIN {X 0,Y 91.597,Z 1037.175,A -85,B 0,C 180,E1 5646.178,E2 5646.178} C_VEL
LIN {X 0,Y 96.445,Z 1032.181,A -85,B 0,C 180,E1 5632.29,E2 5632.29} C_VEL
LIN {X 0,Y 105.317,Z 1025.751,A -85,B 0,C 180,E1 5620.579,E2 5620.579} C_VEL
LIN {X 0,Y 118.365,Z 1016.996,A -85,B 0,C 180,E1 5610.452,E2 5610.452} C_VEL
LIN {X 0,Y 133.42,Z 1006.826,A -85,B 0,C 180,E1 5602.813,E2 5602.813} C_VEL
LIN {X 0,Y 149.543,Z 995.317,A -85,B 0,C 180,E1 5597.036,E2 5597.036} C_VEL
LIN {X 0,Y 166.005,Z 982.435,A -85,B 0,C 180,E1 5592.645,E2 5592.645} C_VEL
LIN {X 0,Y 182.362,Z 968.281,A -85,B 0,C 180,E1 5589.279,E2 5589.279} C_VEL
LIN {X 0,Y 198.307,Z 952.962,A -85,B 0,C 180,E1 5586.647,E2 5586.647} C_VEL
LIN {X 0,Y 213.169,Z 936.841,A -85,B 0,C 180,E1 5584.635,E2 5584.635} C_VEL
LIN {X 0,Y 227.298,Z 919.475,A -85,B 0,C 180,E1 5583.025,E2 5583.025} C_VEL
LIN {X 0,Y 240.458,Z 901.102,A -85,B 0,C 180,E1 5581.753,E2 5581.753} C_VEL
LIN {X 0,Y 252.273,Z 881.918,A -85,B 0,C 180,E1 5580.762,E2 5580.762} C_VEL
LIN {X 0,Y 262.965,Z 861.524,A -85,B 0,C 180,E1 5579.977,E2 5579.977} C_VEL
LIN {X 0,Y 272.28,Z 840.278,A -85,B 0,C 180,E1 5579.387,E2 5579.387} C_VEL
LIN {X 0,Y 280.013,Z 818.338,A -85,B 0,C 180,E1 5578.92,E2 5578.92} C_VEL
LIN {X 0,Y 285.953,Z 795.992,A -85,B 0,C 180,E1 5578.512,E2 5578.512} C_VEL
LIN {X 0,Y 290.368,Z 772.202,A -85,B 0,C 180,E1 5578.119,E2 5578.119} C_VEL
LIN {X 0,Y 303.531,Z 664.138,A -85,B 0,C 180,E1 5576.446,E2 5576.446} C_VEL
LIN {X 0,Y 303.423,Z 664.152,A -85,B 0,C 180,E1 5574.073,E2 5574.073} C_VEL
LIN {X 0,Y 290.082,Z 773.15,A -85,B 0,C 180,E1 5572.503,E2 5572.503} C_VEL
LIN {X 0,Y 285.818,Z 794.948,A -85,B 0,C 180,E1 5572.029,E2 5572.029} C_VEL
LIN {X 0,Y 280.086,Z 816.048,A -85,B 0,C 180,E1 5571.436,E2 5571.436} C_VEL
LIN {X 0,Y 273.068,Z 835.927,A -85,B 0,C 180,E1 5570.728,E2 5570.728} C_VEL
LIN {X 0,Y 264.596,Z 855.306,A -85,B 0,C 180,E1 5569.863,E2 5569.863} C_VEL
LIN {X 0,Y 254.804,Z 874.097,A -85,B 0,C 180,E1 5568.818,E2 5568.818} C_VEL
LIN {X 0,Y 243.689,Z 892.019,A -85,B 0,C 180,E1 5567.561,E2 5567.561} C_VEL
LIN {X 0,Y 231.303,Z 909.153,A -85,B 0,C 180,E1 5566.039,E2 5566.039} C_VEL
LIN {X 0,Y 218.17,Z 924.965,A -85,B 0,C 180,E1 5564.243,E2 5564.243} C_VEL
LIN {X 0,Y 203.567,Z 940.149,A -85,B 0,C 180,E1 5561.974,E2 5561.974} C_VEL
LIN {X 0,Y 188.245,Z 953.989,A -85,B 0,C 180,E1 5559.201,E2 5559.201} C_VEL
LIN {X 0,Y 172.236,Z 966.627,A -85,B 0,C 180,E1 5555.702,E2 5555.702} C_VEL
LIN {X 0,Y 156.923,Z 977.241,A -85,B 0,C 180,E1 5551.558,E2 5551.558} C_VEL
LIN {X 0,Y 141.759,Z 986.35,A -85,B 0,C 180,E1 5546.334,E2 5546.334} C_VEL
LIN {X 0,Y 127.269,Z 994.058,A -85,B 0,C 180,E1 5539.647,E2 5539.647} C_VEL
LIN {X 0,Y 114.484,Z 1000.147,A -85,B 0,C 180,E1 5531.313,E2 5531.313} C_VEL
LIN {X 0,Y 104.231,Z 1004.536,A -85,B 0,C 180,E1 5521.199,E2 5521.199} C_VEL
LIN {X 0,Y 97.172,Z 1007.349,A -85,B 0,C 180,E1 5509.225,E2 5509.225} C_VEL
LIN {X 0,Y 93.88,Z 1008.695,A -85,B 0,C 180,E1 5496.728,E2 5496.728} C_VEL
LIN {X 0,Y 93.667,Z 1008.754,A -85,B 0,C 180,E1 5485.101,E2 5485.101} C_VEL
LIN {X 0,Y 96.69,Z 1007.584,A -85,B 0,C 180,E1 5471.927,E2 5471.927} C_VEL
LIN {X 0,Y 103.395,Z 1004.963,A -85,B 0,C 180,E1 5459.811,E2 5459.811} C_VEL
LIN {X 0,Y 113.572,Z 1000.597,A -85,B 0,C 180,E1 5449.347,E2 5449.347} C_VEL
LIN {X 0,Y 126.549,Z 994.507,A -85,B 0,C 180,E1 5440.668,E2 5440.668} C_VEL
LIN {X 0,Y 140.96,Z 986.93,A -85,B 0,C 180,E1 5433.91,E2 5433.91} C_VEL
LIN {X 0,Y 156.058,Z 977.906,A -85,B 0,C 180,E1 5428.626,E2 5428.626} C_VEL
LIN {X 0,Y 171.333,Z 967.433,A -85,B 0,C 180,E1 5424.441,E2 5424.441} C_VEL
LIN {X 0,Y 187.312,Z 954.971,A -85,B 0,C 180,E1 5420.91,E2 5420.91} C_VEL
LIN {X 0,Y 202.089,Z 941.853,A -85,B 0,C 180,E1 5418.204,E2 5418.204} C_VEL
LIN {X 0,Y 216.3,Z 927.241,A -85,B 0,C 180,E1 5415.951,E2 5415.951} C_VEL
LIN {X 0,Y 230.327,Z 910.721,A -85,B 0,C 180,E1 5414.015,E2 5414.015} C_VEL
LIN {X 0,Y 242.708,Z 893.922,A -85,B 0,C 180,E1 5412.486,E2 5412.486} C_VEL
LIN {X 0,Y 253.815,Z 876.196,A -85,B 0,C 180,E1 5411.216,E2 5411.216} C_VEL
LIN {X 0,Y 264.074,Z 856.927,A -85,B 0,C 180,E1 5410.12,E2 5410.12} C_VEL
LIN {X 0,Y 272.517,Z 838.071,A -85,B 0,C 180,E1 5409.262,E2 5409.262} C_VEL
LIN {X 0,Y 279.803,Z 817.71,A -85,B 0,C 180,E1 5408.523,E2 5408.523} C_VEL
LIN {X 0,Y 285.893,Z 795.756,A -85,B 0,C 180,E1 5407.898,E2 5407.898} C_VEL
LIN {X 0,Y 290.22,Z 774.043,A -85,B 0,C 180,E1 5407.42,E2 5407.42} C_VEL
LIN {X 0,Y 298.38,Z 707.981,A -85,B 0,C 180,E1 5406.443,E2 5406.443} C_VEL
LIN {X 0,Y 303.703,Z 664.183,A -85,B 0,C 180,E1 5405.816,E2 5405.816} C_VEL
LIN {X 0,Y 303.791,Z 664.542,A -85,B 0,C 180,E1 5403.522,E2 5403.522} C_VEL
LIN {X 0,Y 289.864,Z 777.513,A -85,B 0,C 180,E1 5401.801,E2 5401.801} C_VEL
LIN {X 0,Y 285.246,Z 800.085,A -85,B 0,C 180,E1 5401.42,E2 5401.42} C_VEL
LIN {X 0,Y 278.755,Z 822.923,A -85,B 0,C 180,E1 5400.992,E2 5400.992} C_VEL
LIN {X 0,Y 270.975,Z 844.193,A -85,B 0,C 180,E1 5400.521,E2 5400.521} C_VEL
LIN {X 0,Y 261.569,Z 864.942,A -85,B 0,C 180,E1 5399.916,E2 5399.916} C_VEL
LIN {X 0,Y 250.995,Z 884.504,A -85,B 0,C 180,E1 5399.13,E2 5399.13} C_VEL
LIN {X 0,Y 250.309,Z 885.673,A -85,B 0,C 180,E1 5399.076,E2 5399.076} C_VEL
LIN {X 0,Y 246.207,Z 892.269,A -85,B 0,C 180,E1 5398.986,E2 5398.986} C_VEL
LIN {X 0,Y 234.464,Z 908.464,A -85,B 0,C 180,E1 5399.495,E2 5399.495} C_VEL
LIN {X 0,Y 229.751,Z 914.575,A -85,B 0,C 180,E1 5399.334,E2 5399.334} C_VEL
LIN {X 0,Y 215.609,Z 932.129,A -85,B 0,C 180,E1 5397.951,E2 5397.951} C_VEL
LIN {X 0,Y 200.42,Z 948.61,A -85,B 0,C 180,E1 5396.174,E2 5396.174} C_VEL
LIN {X 0,Y 183.397,Z 964.965,A -85,B 0,C 180,E1 5393.741,E2 5393.741} C_VEL
LIN {X 0,Y 166.192,Z 979.645,A -85,B 0,C 180,E1 5390.637,E2 5390.637} C_VEL
LIN {X 0,Y 149.017,Z 992.629,A -85,B 0,C 180,E1 5386.634,E2 5386.634} C_VEL
LIN {X 0,Y 131.142,Z 1004.885,A -85,B 0,C 180,E1 5380.981,E2 5380.981} C_VEL
LIN {X 0,Y 114.934,Z 1015.171,A -85,B 0,C 180,E1 5373.643,E2 5373.643} C_VEL
LIN {X 0,Y 101.123,Z 1023.577,A -85,B 0,C 180,E1 5364.172,E2 5364.172} C_VEL
LIN {X 0,Y 90.282,Z 1030.48,A -85,B 0,C 180,E1 5351.643,E2 5351.643} C_VEL
LIN {X 0,Y 84.183,Z 1035.579,A -85,B 0,C 180,E1 5336.83,E2 5336.83} C_VEL
LIN {X 0,Y 83.039,Z 1038.293,A -85,B 0,C 180,E1 5323.935,E2 5323.935} C_VEL
LIN {X 0,Y 84.045,Z 1039.478,A -85,B 0,C 180,E1 5314.093,E2 5314.093} C_VEL
LIN {X 0,Y 84.478,Z 1039.701,A -85,B 0,C 180,E1 5309.322,E2 5309.322} C_VEL
LIN {X 0,Y 83.402,Z 1039.059,A -85,B 0,C 180,E1 5301.034,E2 5301.034} C_VEL
LIN {X 0,Y 83.465,Z 1036.549,A -85,B 0,C 180,E1 5287.275,E2 5287.275} C_VEL
LIN {X 0,Y 87.774,Z 1032.324,A -85,B 0,C 180,E1 5272.861,E2 5272.861} C_VEL
LIN {X 0,Y 97.052,Z 1026.008,A -85,B 0,C 180,E1 5259.696,E2 5259.696} C_VEL
LIN {X 0,Y 110.706,Z 1017.657,A -85,B 0,C 180,E1 5248.827,E2 5248.827} C_VEL
LIN {X 0,Y 126.311,Z 1007.987,A -85,B 0,C 180,E1 5240.92,E2 5240.92} C_VEL
LIN {X 0,Y 143.343,Z 996.542,A -85,B 0,C 180,E1 5234.955,E2 5234.955} C_VEL
LIN {X 0,Y 160.678,Z 983.746,A -85,B 0,C 180,E1 5230.515,E2 5230.515} C_VEL
LIN {X 0,Y 177.396,Z 970.12,A -85,B 0,C 180,E1 5227.253,E2 5227.253} C_VEL
LIN {X 0,Y 193.632,Z 955.191,A -85,B 0,C 180,E1 5224.723,E2 5224.723} C_VEL
LIN {X 0,Y 209.34,Z 938.905,A -85,B 0,C 180,E1 5222.737,E2 5222.737} C_VEL
LIN {X 0,Y 224.019,Z 921.698,A -85,B 0,C 180,E1 5221.189,E2 5221.189} C_VEL
LIN {X 0,Y 237.373,Z 903.694,A -85,B 0,C 180,E1 5219.999,E2 5219.999} C_VEL
LIN {X 0,Y 249.338,Z 885.093,A -85,B 0,C 180,E1 5219.08,E2 5219.08} C_VEL
LIN {X 0,Y 260.382,Z 865.137,A -85,B 0,C 180,E1 5218.344,E2 5218.344} C_VEL
LIN {X 0,Y 269.661,Z 844.993,A -85,B 0,C 180,E1 5217.812,E2 5217.812} C_VEL
LIN {X 0,Y 277.754,Z 823.452,A -85,B 0,C 180,E1 5217.376,E2 5217.376} C_VEL
LIN {X 0,Y 284.26,Z 801.295,A -85,B 0,C 180,E1 5216.992,E2 5216.992} C_VEL
LIN {X 0,Y 289.045,Z 778.715,A -85,B 0,C 180,E1 5216.635,E2 5216.635} C_VEL
LIN {X 0,Y 294.272,Z 738.687,A -85,B 0,C 180,E1 5216.044,E2 5216.044} C_VEL
LIN {X 0,Y 300.59,Z 686.993,A -85,B 0,C 180,E1 5215.285,E2 5215.285} C_VEL
LIN {X 0,Y 289.719,Z 774.006,A -85,B 0,C 180,E1 5214.074,E2 5214.074} C_VEL
LIN {X 0,Y 285.354,Z 795.865,A -85,B 0,C 180,E1 5213.621,E2 5213.621} C_VEL
LIN {X 0,Y 279.512,Z 816.999,A -85,B 0,C 180,E1 5213.058,E2 5213.058} C_VEL
LIN {X 0,Y 272.364,Z 836.945,A -85,B 0,C 180,E1 5212.389,E2 5212.389} C_VEL
LIN {X 0,Y 263.401,Z 857.058,A -85,B 0,C 180,E1 5211.541,E2 5211.541} C_VEL
LIN {X 0,Y 252.961,Z 876.538,A -85,B 0,C 180,E1 5210.51,E2 5210.51} C_VEL
LIN {X 0,Y 241.188,Z 895.076,A -85,B 0,C 180,E1 5209.267,E2 5209.267} C_VEL
LIN {X 0,Y 228.146,Z 912.453,A -85,B 0,C 180,E1 5207.773,E2 5207.773} C_VEL
LIN {X 0,Y 213.667,Z 929.096,A -85,B 0,C 180,E1 5205.916,E2 5205.916} C_VEL
LIN {X 0,Y 198.932,Z 943.807,A -85,B 0,C 180,E1 5203.74,E2 5203.74} C_VEL
LIN {X 0,Y 183.834,Z 956.87,A -85,B 0,C 180,E1 5201.152,E2 5201.152} C_VEL
LIN {X 0,Y 167.439,Z 969.22,A -85,B 0,C 180,E1 5197.757,E2 5197.757} C_VEL
LIN {X 0,Y 150.873,Z 980.077,A -85,B 0,C 180,E1 5193.466,E2 5193.466} C_VEL
LIN {X 0,Y 135.262,Z 989.002,A -85,B 0,C 180,E1 5188.222,E2 5188.222} C_VEL
LIN {X 0,Y 120.241,Z 996.399,A -85,B 0,C 180,E1 5181.413,E2 5181.413} C_VEL
LIN {X 0,Y 106.603,Z 1002.331,A -85,B 0,C 180,E1 5172.479,E2 5172.479} C_VEL
LIN {X 0,Y 95.834,Z 1006.551,A -85,B 0,C 180,E1 5161.444,E2 5161.444} C_VEL
LIN {X 0,Y 88.76,Z 1009.103,A -85,B 0,C 180,E1 5148.386,E2 5148.386} C_VEL
LIN {X 0,Y 85.763,Z 1010.128,A -85,B 0,C 180,E1 5134.681,E2 5134.681} C_VEL
LIN {X 0,Y 86.135,Z 1010.055,A -85,B 0,C 180,E1 5121.993,E2 5121.993} C_VEL
LIN {X 0,Y 89.981,Z 1008.666,A -85,B 0,C 180,E1 5108.488,E2 5108.488} C_VEL
LIN {X 0,Y 98.085,Z 1005.741,A -85,B 0,C 180,E1 5095.663,E2 5095.663} C_VEL
LIN {X 0,Y 109.416,Z 1001.295,A -85,B 0,C 180,E1 5085.28,E2 5085.28} C_VEL
LIN {X 0,Y 122.906,Z 995.238,A -85,B 0,C 180,E1 5077.132,E2 5077.132} C_VEL
LIN {X 0,Y 138.98,Z 987.041,A -85,B 0,C 180,E1 5070.309,E2 5070.309} C_VEL
LIN {X 0,Y 154.87,Z 977.764,A -85,B 0,C 180,E1 5065.329,E2 5065.329} C_VEL
LIN {X 0,Y 170.772,Z 967.042,A -85,B 0,C 180,E1 5061.418,E2 5061.418} C_VEL
LIN {X 0,Y 186.402,Z 954.932,A -85,B 0,C 180,E1 5058.298,E2 5058.298} C_VEL
LIN {X 0,Y 201.565,Z 941.565,A -85,B 0,C 180,E1 5055.775,E2 5055.775} C_VEL
LIN {X 0,Y 216.106,Z 926.779,A -85,B 0,C 180,E1 5053.684,E2 5053.684} C_VEL
LIN {X 0,Y 229.943,Z 910.512,A -85,B 0,C 180,E1 5051.938,E2 5051.938} C_VEL
LIN {X 0,Y 243.007,Z 892.729,A -85,B 0,C 180,E1 5050.461,E2 5050.461} C_VEL
LIN {X 0,Y 254.451,Z 874.511,A -85,B 0,C 180,E1 5049.272,E2 5049.272} C_VEL
LIN {X 0,Y 264.238,Z 855.887,A -85,B 0,C 180,E1 5048.308,E2 5048.308} C_VEL
LIN {X 0,Y 273.274,Z 835.266,A -85,B 0,C 180,E1 5047.455,E2 5047.455} C_VEL
LIN {X 0,Y 280.431,Z 815.049,A -85,B 0,C 180,E1 5046.791,E2 5046.791} C_VEL
LIN {X 0,Y 286.096,Z 793.866,A -85,B 0,C 180,E1 5046.242,E2 5046.242} C_VEL
LIN {X 0,Y 290.438,Z 770.886,A -85,B 0,C 180,E1 5045.779,E2 5045.779} C_VEL
LIN {X 0,Y 300.486,Z 690.183,A -85,B 0,C 180,E1 5044.663,E2 5044.663} C_VEL
LIN {X 0,Y 289.594,Z 777.129,A -85,B 0,C 180,E1 5043.392,E2 5043.392} C_VEL
LIN {X 0,Y 284.863,Z 799.859,A -85,B 0,C 180,E1 5043.034,E2 5043.034} C_VEL
LIN {X 0,Y 278.54,Z 821.867,A -85,B 0,C 180,E1 5042.657,E2 5042.657} C_VEL
LIN {X 0,Y 270.875,Z 842.775,A -85,B 0,C 180,E1 5042.246,E2 5042.246} C_VEL
LIN {X 0,Y 261.584,Z 863.169,A -85,B 0,C 180,E1 5041.723,E2 5041.723} C_VEL
LIN {X 0,Y 250.504,Z 883.546,A -85,B 0,C 180,E1 5040.992,E2 5040.992} C_VEL
LIN {X 0,Y 238.468,Z 902.499,A -85,B 0,C 180,E1 5040.079,E2 5040.079} C_VEL
LIN {X 0,Y 229.751,Z 914.575,A -85,B 0,C 180,E1 5039.334,E2 5039.334} C_VEL
LIN {X 0,Y 224.856,Z 920.713,A -85,B 0,C 180,E1 5039.144,E2 5039.144} C_VEL
LIN {X 0,Y 211.262,Z 935.442,A -85,B 0,C 180,E1 5039.495,E2 5039.495} C_VEL
LIN {X 0,Y 206.003,Z 940.943,A -85,B 0,C 180,E1 5039.249,E2 5039.249} C_VEL
LIN {X 0,Y 190.168,Z 956.594,A -85,B 0,C 180,E1 5037.413,E2 5037.413} C_VEL
LIN {X 0,Y 172.665,Z 971.944,A -85,B 0,C 180,E1 5034.882,E2 5034.882} C_VEL
LIN {X 0,Y 154.657,Z 985.917,A -85,B 0,C 180,E1 5031.553,E2 5031.553} C_VEL
LIN {X 0,Y 136.453,Z 998.396,A -85,B 0,C 180,E1 5027.049,E2 5027.049} C_VEL
LIN {X 0,Y 118.286,Z 1009.633,A -85,B 0,C 180,E1 5020.753,E2 5020.753} C_VEL
LIN {X 0,Y 102.47,Z 1018.716,A -85,B 0,C 180,E1 5012.616,E2 5012.616} C_VEL
LIN {X 0,Y 89.154,Z 1026.1,A -85,B 0,C 180,E1 5001.725,E2 5001.725} C_VEL
LIN {X 0,Y 79.438,Z 1032.016,A -85,B 0,C 180,E1 4987.168,E2 4987.168} C_VEL
LIN {X 0,Y 75.391,Z 1035.855,A -85,B 0,C 180,E1 4971.799,E2 4971.799} C_VEL
LIN {X 0,Y 75.641,Z 1037.854,A -85,B 0,C 180,E1 4957.544,E2 4957.544} C_VEL
LIN {X 0,Y 76.622,Z 1038.36,A -85,B 0,C 180,E1 4950,E2 4950} C_VEL
LIN {X 0,Y 75.546,Z 1037.783,A -85,B 0,C 180,E1 4941.629,E2 4941.629} C_VEL
LIN {X 0,Y 75.581,Z 1035.491,A -85,B 0,C 180,E1 4926.617,E2 4926.617} C_VEL
LIN {X 0,Y 79.768,Z 1031.759,A -85,B 0,C 180,E1 4912.106,E2 4912.106} C_VEL
LIN {X 0,Y 90.275,Z 1025.4,A -85,B 0,C 180,E1 4897.112,E2 4897.112} C_VEL
LIN {X 0,Y 103.9,Z 1017.867,A -85,B 0,C 180,E1 4886.495,E2 4886.495} C_VEL
LIN {X 0,Y 120.357,Z 1008.329,A -85,B 0,C 180,E1 4878.4,E2 4878.4} C_VEL
LIN {X 0,Y 137.747,Z 997.414,A -85,B 0,C 180,E1 4872.576,E2 4872.576} C_VEL
LIN {X 0,Y 155.587,Z 985.064,A -85,B 0,C 180,E1 4868.244,E2 4868.244} C_VEL
LIN {X 0,Y 173.651,Z 970.983,A -85,B 0,C 180,E1 4864.954,E2 4864.954} C_VEL
LIN {X 0,Y 190.168,Z 956.388,A -85,B 0,C 180,E1 4862.579,E2 4862.579} C_VEL
LIN {X 0,Y 206.488,Z 940.164,A -85,B 0,C 180,E1 4860.693,E2 4860.693} C_VEL
LIN {X 0,Y 220.987,Z 923.733,A -85,B 0,C 180,E1 4859.297,E2 4859.297} C_VEL
LIN {X 0,Y 235.09,Z 905.379,A -85,B 0,C 180,E1 4858.158,E2 4858.158} C_VEL
LIN {X 0,Y 248.252,Z 885.543,A -85,B 0,C 180,E1 4857.257,E2 4857.257} C_VEL
LIN {X 0,Y 259.423,Z 865.818,A -85,B 0,C 180,E1 4856.599,E2 4856.599} C_VEL
LIN {X 0,Y 269.083,Z 845.202,A -85,B 0,C 180,E1 4856.113,E2 4856.113} C_VEL
LIN {X 0,Y 277.394,Z 823.503,A -85,B 0,C 180,E1 4855.723,E2 4855.723} C_VEL
LIN {X 0,Y 283.97,Z 801.588,A -85,B 0,C 180,E1 4855.38,E2 4855.38} C_VEL
LIN {X 0,Y 285.626,Z 794.64,A -85,B 0,C 180,E1 4855.263,E2 4855.263} C_VEL
LIN {X 0,Y 279.889,Z 815.799,A -85,B 0,C 180,E1 4854.747,E2 4854.747} C_VEL
LIN {X 0,Y 272.368,Z 836.731,A -85,B 0,C 180,E1 4854.1,E2 4854.1} C_VEL
LIN {X 0,Y 263.397,Z 856.863,A -85,B 0,C 180,E1 4853.319,E2 4853.319} C_VEL
LIN {X 0,Y 253.194,Z 875.948,A -85,B 0,C 180,E1 4852.394,E2 4852.394} C_VEL
LIN {X 0,Y 241.75,Z 893.893,A -85,B 0,C 180,E1 4851.299,E2 4851.299} C_VEL
LIN {X 0,Y 228.454,Z 911.715,A -85,B 0,C 180,E1 4849.917,E2 4849.917} C_VEL
LIN {X 0,Y 214.434,Z 927.928,A -85,B 0,C 180,E1 4848.292,E2 4848.292} C_VEL
LIN {X 0,Y 199.624,Z 942.721,A -85,B 0,C 180,E1 4846.337,E2 4846.337} C_VEL
LIN {X 0,Y 183.53,Z 956.601,A -85,B 0,C 180,E1 4843.867,E2 4843.867} C_VEL
LIN {X 0,Y 166.356,Z 969.426,A -85,B 0,C 180,E1 4840.671,E2 4840.671} C_VEL
LIN {X 0,Y 149.656,Z 980.232,A -85,B 0,C 180,E1 4836.784,E2 4836.784} C_VEL
LIN {X 0,Y 132.835,Z 989.544,A -85,B 0,C 180,E1 4831.724,E2 4831.724} C_VEL
LIN {X 0,Y 116.901,Z 997.138,A -85,B 0,C 180,E1 4825.195,E2 4825.195} C_VEL
LIN {X 0,Y 102.114,Z 1003.258,A -85,B 0,C 180,E1 4816.434,E2 4816.434} C_VEL
LIN {X 0,Y 90.098,Z 1007.641,A -85,B 0,C 180,E1 4805.245,E2 4805.245} C_VEL
LIN {X 0,Y 81.83,Z 1010.281,A -85,B 0,C 180,E1 4791.504,E2 4791.504} C_VEL
LIN {X 0,Y 77.976,Z 1011.477,A -85,B 0,C 180,E1 4775.888,E2 4775.888} C_VEL
LIN {X 0,Y 78.128,Z 1011.452,A -85,B 0,C 180,E1 4762.647,E2 4762.647} C_VEL
LIN {X 0,Y 82.373,Z 1010.129,A -85,B 0,C 180,E1 4747.144,E2 4747.144} C_VEL
LIN {X 0,Y 90.999,Z 1007.354,A -85,B 0,C 180,E1 4733.606,E2 4733.606} C_VEL
LIN {X 0,Y 103.297,Z 1002.891,A -85,B 0,C 180,E1 4722.639,E2 4722.639} C_VEL
LIN {X 0,Y 117.559,Z 996.931,A -85,B 0,C 180,E1 4714.411,E2 4714.411} C_VEL
LIN {X 0,Y 133.561,Z 989.27,A -85,B 0,C 180,E1 4707.948,E2 4707.948} C_VEL
LIN {X 0,Y 149.965,Z 980.189,A -85,B 0,C 180,E1 4703.06,E2 4703.06} C_VEL
LIN {X 0,Y 166.291,Z 969.626,A -85,B 0,C 180,E1 4699.266,E2 4699.266} C_VEL
LIN {X 0,Y 183.176,Z 957.086,A -85,B 0,C 180,E1 4696.117,E2 4696.117} C_VEL
LIN {X 0,Y 198.651,Z 943.9,A -85,B 0,C 180,E1 4693.73,E2 4693.73} C_VEL
LIN {X 0,Y 213.448,Z 929.225,A -85,B 0,C 180,E1 4691.755,E2 4691.755} C_VEL
LIN {X 0,Y 227.978,Z 912.639,A -85,B 0,C 180,E1 4690.063,E2 4690.063} C_VEL
LIN {X 0,Y 240.758,Z 895.781,A -85,B 0,C 180,E1 4688.731,E2 4688.731} C_VEL
LIN {X 0,Y 252.197,Z 878.03,A -85,B 0,C 180,E1 4687.625,E2 4687.625} C_VEL
LIN {X 0,Y 262.743,Z 858.734,A -85,B 0,C 180,E1 4686.669,E2 4686.669} C_VEL
LIN {X 0,Y 271.841,Z 838.791,A -85,B 0,C 180,E1 4685.88,E2 4685.88} C_VEL
LIN {X 0,Y 279.133,Z 818.851,A -85,B 0,C 180,E1 4685.248,E2 4685.248} C_VEL
LIN {X 0,Y 285.328,Z 797.025,A -85,B 0,C 180,E1 4684.688,E2 4684.688} C_VEL
LIN {X 0,Y 278.76,Z 820.211,A -85,B 0,C 180,E1 4684.333,E2 4684.333} C_VEL
LIN {X 0,Y 271.116,Z 841.129,A -85,B 0,C 180,E1 4683.973,E2 4683.973} C_VEL
LIN {X 0,Y 261.454,Z 862.227,A -85,B 0,C 180,E1 4683.503,E2 4683.503} C_VEL
LIN {X 0,Y 250.278,Z 882.59,A -85,B 0,C 180,E1 4682.858,E2 4682.858} C_VEL
LIN {X 0,Y 238.12,Z 901.517,A -85,B 0,C 180,E1 4682.047,E2 4682.047} C_VEL
LIN {X 0,Y 224.854,Z 919.261,A -85,B 0,C 180,E1 4681.02,E2 4681.02} C_VEL
LIN {X 0,Y 209.976,Z 936.62,A -85,B 0,C 180,E1 4679.655,E2 4679.655} C_VEL
LIN {X 0,Y 206.003,Z 940.943,A -85,B 0,C 180,E1 4679.249,E2 4679.249} C_VEL
LIN {X 0,Y 200.569,Z 946.407,A -85,B 0,C 180,E1 4678.967,E2 4678.967} C_VEL
LIN {X 0,Y 185.282,Z 959.556,A -85,B 0,C 180,E1 4679.109,E2 4679.109} C_VEL
LIN {X 0,Y 179.4,Z 964.372,A -85,B 0,C 180,E1 4678.705,E2 4678.705} C_VEL
LIN {X 0,Y 161.359,Z 978.745,A -85,B 0,C 180,E1 4676.064,E2 4676.064} C_VEL
LIN {X 0,Y 143.176,Z 991.539,A -85,B 0,C 180,E1 4672.592,E2 4672.592} C_VEL
LIN {X 0,Y 124.789,Z 1002.948,A -85,B 0,C 180,E1 4667.828,E2 4667.828} C_VEL
LIN {X 0,Y 105.94,Z 1013.472,A -85,B 0,C 180,E1 4660.7,E2 4660.7} C_VEL
LIN {X 0,Y 90.04,Z 1021.696,A -85,B 0,C 180,E1 4651.314,E2 4651.314} C_VEL
LIN {X 0,Y 77.367,Z 1028.084,A -85,B 0,C 180,E1 4638.553,E2 4638.553} C_VEL
LIN {X 0,Y 69.164,Z 1033.033,A -85,B 0,C 180,E1 4621.361,E2 4621.361} C_VEL
LIN {X 0,Y 67.18,Z 1035.685,A -85,B 0,C 180,E1 4605.539,E2 4605.539} C_VEL
LIN {X 0,Y 68.395,Z 1036.863,A -85,B 0,C 180,E1 4592.513,E2 4592.513} C_VEL
LIN {X 0,Y 68.655,Z 1036.96,A -85,B 0,C 180,E1 4589.165,E2 4589.165} C_VEL
LIN {X 0,Y 67.247,Z 1036.022,A -85,B 0,C 180,E1 4577.113,E2 4577.113} C_VEL
LIN {X 0,Y 68.564,Z 1033.492,A -85,B 0,C 180,E1 4561.035,E2 4561.035} C_VEL
LIN {X 0,Y 75.442,Z 1029.139,A -85,B 0,C 180,E1 4544.3,E2 4544.3} C_VEL
LIN {X 0,Y 87.34,Z 1022.943,A -85,B 0,C 180,E1 4530.84,E2 4530.84} C_VEL
LIN {X 0,Y 103.935,Z 1014.443,A -85,B 0,C 180,E1 4520.261,E2 4520.261} C_VEL
LIN {X 0,Y 121.238,Z 1004.973,A -85,B 0,C 180,E1 4513.303,E2 4513.303} C_VEL
LIN {X 0,Y 139.435,Z 993.821,A -85,B 0,C 180,E1 4508.244,E2 4508.244} C_VEL
LIN {X 0,Y 157.483,Z 981.419,A -85,B 0,C 180,E1 4504.586,E2 4504.586} C_VEL
LIN {X 0,Y 175.07,Z 967.873,A -85,B 0,C 180,E1 4501.869,E2 4501.869} C_VEL
LIN {X 0,Y 191.976,Z 953.008,A -85,B 0,C 180,E1 4499.803,E2 4499.803} C_VEL
LIN {X 0,Y 208.592,Z 936.389,A -85,B 0,C 180,E1 4498.166,E2 4498.166} C_VEL
LIN {X 0,Y 223.282,Z 919.666,A -85,B 0,C 180,E1 4496.974,E2 4496.974} C_VEL
LIN {X 0,Y 236.526,Z 902.28,A -85,B 0,C 180,E1 4496.065,E2 4496.065} C_VEL
LIN {X 0,Y 249.299,Z 882.881,A -85,B 0,C 180,E1 4495.319,E2 4495.319} C_VEL
LIN {X 0,Y 259.83,Z 864.292,A -85,B 0,C 180,E1 4494.79,E2 4494.79} C_VEL
LIN {X 0,Y 248.891,Z 883.141,A -85,B 0,C 180,E1 4493.87,E2 4493.87} C_VEL
LIN {X 0,Y 235.88,Z 902.162,A -85,B 0,C 180,E1 4492.702,E2 4492.702} C_VEL
LIN {X 0,Y 222.482,Z 918.954,A -85,B 0,C 180,E1 4491.384,E2 4491.384} C_VEL
LIN {X 0,Y 208.248,Z 934.262,A -85,B 0,C 180,E1 4489.826,E2 4489.826} C_VEL
LIN {X 0,Y 192.308,Z 949.098,A -85,B 0,C 180,E1 4487.814,E2 4487.814} C_VEL
LIN {X 0,Y 175.694,Z 962.493,A -85,B 0,C 180,E1 4485.344,E2 4485.344} C_VEL
LIN {X 0,Y 158.549,Z 974.407,A -85,B 0,C 180,E1 4482.225,E2 4482.225} C_VEL
LIN {X 0,Y 141.053,Z 984.768,A -85,B 0,C 180,E1 4478.218,E2 4478.218} C_VEL
LIN {X 0,Y 123.557,Z 993.646,A -85,B 0,C 180,E1 4472.894,E2 4472.894} C_VEL
LIN {X 0,Y 107.309,Z 1000.709,A -85,B 0,C 180,E1 4466.008,E2 4466.008} C_VEL
LIN {X 0,Y 92.329,Z 1006.21,A -85,B 0,C 180,E1 4456.516,E2 4456.516} C_VEL
LIN {X 0,Y 80.328,Z 1009.98,A -85,B 0,C 180,E1 4444.065,E2 4444.065} C_VEL
LIN {X 0,Y 72.582,Z 1012.198,A -85,B 0,C 180,E1 4428.472,E2 4428.472} C_VEL
LIN {X 0,Y 69.887,Z 1012.916,A -85,B 0,C 180,E1 4413.281,E2 4413.281} C_VEL
LIN {X 0,Y 71.296,Z 1012.552,A -85,B 0,C 180,E1 4396.207,E2 4396.207} C_VEL
LIN {X 0,Y 77.325,Z 1010.933,A -85,B 0,C 180,E1 4380.57,E2 4380.57} C_VEL
LIN {X 0,Y 88.072,Z 1007.639,A -85,B 0,C 180,E1 4367.065,E2 4367.065} C_VEL
LIN {X 0,Y 102.927,Z 1002.441,A -85,B 0,C 180,E1 4356.265,E2 4356.265} C_VEL
LIN {X 0,Y 118.716,Z 996.007,A -85,B 0,C 180,E1 4348.846,E2 4348.846} C_VEL
LIN {X 0,Y 135.045,Z 988.104,A -85,B 0,C 180,E1 4343.352,E2 4343.352} C_VEL
LIN {X 0,Y 152.293,Z 978.401,A -85,B 0,C 180,E1 4339.017,E2 4339.017} C_VEL
LIN {X 0,Y 169.269,Z 967.358,A -85,B 0,C 180,E1 4335.67,E2 4335.67} C_VEL
LIN {X 0,Y 185.761,Z 954.85,A -85,B 0,C 180,E1 4333.034,E2 4333.034} C_VEL
LIN {X 0,Y 201.612,Z 940.945,A -85,B 0,C 180,E1 4330.902,E2 4330.902} C_VEL
LIN {X 0,Y 216.729,Z 925.699,A -85,B 0,C 180,E1 4329.149,E2 4329.149} C_VEL
LIN {X 0,Y 230.693,Z 909.352,A -85,B 0,C 180,E1 4327.722,E2 4327.722} C_VEL
LIN {X 0,Y 243.547,Z 891.755,A -85,B 0,C 180,E1 4326.528,E2 4326.528} C_VEL
LIN {X 0,Y 255.638,Z 872.327,A -85,B 0,C 180,E1 4325.489,E2 4325.489} C_VEL
LIN {X 0,Y 259.368,Z 865.641,A -85,B 0,C 180,E1 4325.18,E2 4325.18} C_VEL
LIN {X 0,Y 248.315,Z 884.946,A -85,B 0,C 180,E1 4324.62,E2 4324.62} C_VEL
LIN {X 0,Y 235.504,Z 904.044,A -85,B 0,C 180,E1 4323.863,E2 4323.863} C_VEL
LIN {X 0,Y 221.755,Z 921.82,A -85,B 0,C 180,E1 4322.905,E2 4322.905} C_VEL
LIN {X 0,Y 206.793,Z 938.575,A -85,B 0,C 180,E1 4321.663,E2 4321.663} C_VEL
LIN {X 0,Y 189.975,Z 955.05,A -85,B 0,C 180,E1 4319.971,E2 4319.971} C_VEL
LIN {X 0,Y 179.4,Z 964.372,A -85,B 0,C 180,E1 4318.705,E2 4318.705} C_VEL
LIN {X 0,Y 173.416,Z 969.18,A -85,B 0,C 180,E1 4318.254,E2 4318.254} C_VEL
LIN {X 0,Y 156.812,Z 980.514,A -85,B 0,C 180,E1 4318.097,E2 4318.097} C_VEL
LIN {X 0,Y 150.454,Z 984.647,A -85,B 0,C 180,E1 4317.483,E2 4317.483} C_VEL
LIN {X 0,Y 130.796,Z 997.139,A -85,B 0,C 180,E1 4313.606,E2 4313.606} C_VEL
LIN {X 0,Y 112.256,Z 1007.45,A -85,B 0,C 180,E1 4308.456,E2 4308.456} C_VEL
LIN {X 0,Y 93.339,Z 1016.873,A -85,B 0,C 180,E1 4300.505,E2 4300.505} C_VEL
LIN {X 0,Y 76.999,Z 1024.409,A -85,B 0,C 180,E1 4288.985,E2 4288.985} C_VEL
LIN {X 0,Y 65.416,Z 1029.766,A -85,B 0,C 180,E1 4273.457,E2 4273.457} C_VEL
LIN {X 0,Y 59.68,Z 1033.522,A -85,B 0,C 180,E1 4253.709,E2 4253.709} C_VEL
LIN {X 0,Y 59.871,Z 1035.234,A -85,B 0,C 180,E1 4236.713,E2 4236.713} C_VEL
LIN {X 0,Y 60.817,Z 1035.622,A -85,B 0,C 180,E1 4230,E2 4230} C_VEL
LIN {X 0,Y 59.3,Z 1034.718,A -85,B 0,C 180,E1 4216.346,E2 4216.346} C_VEL
LIN {X 0,Y 61.328,Z 1032.081,A -85,B 0,C 180,E1 4197.451,E2 4197.451} C_VEL
LIN {X 0,Y 70.076,Z 1027.512,A -85,B 0,C 180,E1 4178.885,E2 4178.885} C_VEL
LIN {X 0,Y 84.009,Z 1021.132,A -85,B 0,C 180,E1 4165.237,E2 4165.237} C_VEL
LIN {X 0,Y 101.692,Z 1012.74,A -85,B 0,C 180,E1 4155.513,E2 4155.513} C_VEL
LIN {X 0,Y 120.474,Z 1002.929,A -85,B 0,C 180,E1 4149.019,E2 4149.019} C_VEL
LIN {X 0,Y 139.511,Z 991.684,A -85,B 0,C 180,E1 4144.52,E2 4144.52} C_VEL
LIN {X 0,Y 158.021,Z 979.196,A -85,B 0,C 180,E1 4141.324,E2 4141.324} C_VEL
LIN {X 0,Y 177.013,Z 964.648,A -85,B 0,C 180,E1 4138.837,E2 4138.837} C_VEL
LIN {X 0,Y 194.558,Z 949.315,A -85,B 0,C 180,E1 4137.053,E2 4137.053} C_VEL
LIN {X 0,Y 211.085,Z 932.62,A -85,B 0,C 180,E1 4135.693,E2 4135.693} C_VEL
LIN {X 0,Y 226.273,Z 915.015,A -85,B 0,C 180,E1 4134.675,E2 4134.675} C_VEL
LIN {X 0,Y 231.866,Z 907.919,A -85,B 0,C 180,E1 4134.327,E2 4134.327} C_VEL
LIN {X 0,Y 218.06,Z 924.2,A -85,B 0,C 180,E1 4133.08,E2 4133.08} C_VEL
LIN {X 0,Y 202.218,Z 940.342,A -85,B 0,C 180,E1 4131.455,E2 4131.455} C_VEL
LIN {X 0,Y 186.075,Z 954.55,A -85,B 0,C 180,E1 4129.529,E2 4129.529} C_VEL
LIN {X 0,Y 169.208,Z 967.218,A -85,B 0,C 180,E1 4127.162,E2 4127.162} C_VEL
LIN {X 0,Y 151.763,Z 978.538,A -85,B 0,C 180,E1 4124.133,E2 4124.133} C_VEL
LIN {X 0,Y 133.91,Z 988.488,A -85,B 0,C 180,E1 4120.188,E2 4120.188} C_VEL
LIN {X 0,Y 115.98,Z 996.883,A -85,B 0,C 180,E1 4114.851,E2 4114.851} C_VEL
LIN {X 0,Y 98.755,Z 1003.63,A -85,B 0,C 180,E1 4107.545,E2 4107.545} C_VEL
LIN {X 0,Y 82.496,Z 1008.946,A -85,B 0,C 180,E1 4096.653,E2 4096.653} C_VEL
LIN {X 0,Y 70.572,Z 1012.264,A -85,B 0,C 180,E1 4082.574,E2 4082.574} C_VEL
LIN {X 0,Y 63.674,Z 1013.899,A -85,B 0,C 180,E1 4065.483,E2 4065.483} C_VEL
LIN {X 0,Y 61.976,Z 1014.308,A -85,B 0,C 180,E1 4047.226,E2 4047.226} C_VEL
LIN {X 0,Y 64.838,Z 1013.642,A -85,B 0,C 180,E1 4030.168,E2 4030.168} C_VEL
LIN {X 0,Y 73.859,Z 1011.401,A -85,B 0,C 180,E1 4012.47,E2 4012.47} C_VEL
LIN {X 0,Y 87.015,Z 1007.668,A -85,B 0,C 180,E1 3999.657,E2 3999.657} C_VEL
LIN {X 0,Y 103.044,Z 1002.178,A -85,B 0,C 180,E1 3990.278,E2 3990.278} C_VEL
LIN {X 0,Y 120.097,Z 995.151,A -85,B 0,C 180,E1 3983.68,E2 3983.68} C_VEL
LIN {X 0,Y 138.259,Z 986.314,A -85,B 0,C 180,E1 3978.671,E2 3978.671} C_VEL
LIN {X 0,Y 156.268,Z 976.014,A -85,B 0,C 180,E1 3974.948,E2 3974.948} C_VEL
LIN {X 0,Y 173.82,Z 964.129,A -85,B 0,C 180,E1 3972.07,E2 3972.07} C_VEL
LIN {X 0,Y 190.76,Z 950.808,A -85,B 0,C 180,E1 3969.804,E2 3969.804} C_VEL
LIN {X 0,Y 206.01,Z 937.036,A -85,B 0,C 180,E1 3968.065,E2 3968.065} C_VEL
LIN {X 0,Y 220.926,Z 921.349,A -85,B 0,C 180,E1 3966.581,E2 3966.581} C_VEL
LIN {X 0,Y 231.49,Z 908.796,A -85,B 0,C 180,E1 3965.625,E2 3965.625} C_VEL
LIN {X 0,Y 216.7,Z 926.687,A -85,B 0,C 180,E1 3964.7,E2 3964.7} C_VEL
LIN {X 0,Y 200.205,Z 944.044,A -85,B 0,C 180,E1 3963.437,E2 3963.437} C_VEL
LIN {X 0,Y 183.068,Z 959.794,A -85,B 0,C 180,E1 3961.821,E2 3961.821} C_VEL
LIN {X 0,Y 164.952,Z 974.322,A -85,B 0,C 180,E1 3959.654,E2 3959.654} C_VEL
LIN {X 0,Y 150.454,Z 984.647,A -85,B 0,C 180,E1 3957.483,E2 3957.483} C_VEL
LIN {X 0,Y 144.001,Z 988.687,A -85,B 0,C 180,E1 3956.785,E2 3956.785} C_VEL
LIN {X 0,Y 126.252,Z 998.035,A -85,B 0,C 180,E1 3956.083,E2 3956.083} C_VEL
LIN {X 0,Y 119.644,Z 1001.416,A -85,B 0,C 180,E1 3955.107,E2 3955.107} C_VEL
LIN {X 0,Y 99.736,Z 1011.336,A -85,B 0,C 180,E1 3949.252,E2 3949.252} C_VEL
LIN {X 0,Y 80.727,Z 1019.709,A -85,B 0,C 180,E1 3940.274,E2 3940.274} C_VEL
LIN {X 0,Y 65.352,Z 1025.96,A -85,B 0,C 180,E1 3927.296,E2 3927.296} C_VEL
LIN {X 0,Y 54.446,Z 1030.654,A -85,B 0,C 180,E1 3907.302,E2 3907.302} C_VEL
LIN {X 0,Y 51.361,Z 1033.403,A -85,B 0,C 180,E1 3884.659,E2 3884.659} C_VEL
LIN {X 0,Y 52.828,Z 1034.238,A -85,B 0,C 180,E1 3870,E2 3870} C_VEL
LIN {X 0,Y 51.351,Z 1033.174,A -85,B 0,C 180,E1 3853.018,E2 3853.018} C_VEL
LIN {X 0,Y 54.785,Z 1030.452,A -85,B 0,C 180,E1 3831.646,E2 3831.646} C_VEL
LIN {X 0,Y 65.997,Z 1025.638,A -85,B 0,C 180,E1 3811.96,E2 3811.96} C_VEL
LIN {X 0,Y 81.538,Z 1019.323,A -85,B 0,C 180,E1 3799.226,E2 3799.226} C_VEL
LIN {X 0,Y 99.736,Z 1011.246,A -85,B 0,C 180,E1 3790.745,E2 3790.745} C_VEL
LIN {X 0,Y 119.428,Z 1001.426,A -85,B 0,C 180,E1 3784.94,E2 3784.94} C_VEL
LIN {X 0,Y 139.003,Z 990.237,A -85,B 0,C 180,E1 3781.008,E2 3781.008} C_VEL
LIN {X 0,Y 158.303,Z 977.508,A -85,B 0,C 180,E1 3778.189,E2 3778.189} C_VEL
LIN {X 0,Y 178.414,Z 962.269,A -85,B 0,C 180,E1 3775.986,E2 3775.986} C_VEL
LIN {X 0,Y 195.872,Z 947.072,A -85,B 0,C 180,E1 3774.513,E2 3774.513} C_VEL
LIN {X 0,Y 203.961,Z 939.276,A -85,B 0,C 180,E1 3773.936,E2 3773.936} C_VEL
LIN {X 0,Y 187.684,Z 953.591,A -85,B 0,C 180,E1 3772.262,E2 3772.262} C_VEL
LIN {X 0,Y 170.476,Z 966.643,A -85,B 0,C 180,E1 3770.18,E2 3770.18} C_VEL
LIN {X 0,Y 152.542,Z 978.343,A -85,B 0,C 180,E1 3767.507,E2 3767.507} C_VEL
LIN {X 0,Y 134.156,Z 988.5,A -85,B 0,C 180,E1 3764.037,E2 3764.037} C_VEL
LIN {X 0,Y 116.311,Z 996.773,A -85,B 0,C 180,E1 3759.557,E2 3759.557} C_VEL
LIN {X 0,Y 97.692,Z 1004,A -85,B 0,C 180,E1 3752.929,E2 3752.929} C_VEL
LIN {X 0,Y 80.725,Z 1009.422,A -85,B 0,C 180,E1 3743.518,E2 3743.518} C_VEL
LIN {X 0,Y 66.477,Z 1013.047,A -85,B 0,C 180,E1 3729.904,E2 3729.904} C_VEL
LIN {X 0,Y 57.186,Z 1015.043,A -85,B 0,C 180,E1 3711.542,E2 3711.542} C_VEL
LIN {X 0,Y 54.06,Z 1015.706,A -85,B 0,C 180,E1 3691.06,E2 3691.06} C_VEL
LIN {X 0,Y 56.596,Z 1015.175,A -85,B 0,C 180,E1 3670.387,E2 3670.387} C_VEL
LIN {X 0,Y 65.028,Z 1013.464,A -85,B 0,C 180,E1 3652.046,E2 3652.046} C_VEL
LIN {X 0,Y 78.613,Z 1010.018,A -85,B 0,C 180,E1 3637.948,E2 3637.948} C_VEL
LIN {X 0,Y 95.215,Z 1004.919,A -85,B 0,C 180,E1 3628.104,E2 3628.104} C_VEL
LIN {X 0,Y 112.793,Z 998.396,A -85,B 0,C 180,E1 3621.443,E2 3621.443} C_VEL
LIN {X 0,Y 131.392,Z 990.014,A -85,B 0,C 180,E1 3616.496,E2 3616.496} C_VEL
LIN {X 0,Y 149.753,Z 980.112,A -85,B 0,C 180,E1 3612.887,E2 3612.887} C_VEL
LIN {X 0,Y 168.542,Z 968.191,A -85,B 0,C 180,E1 3610.007,E2 3610.007} C_VEL
LIN {X 0,Y 185.733,Z 955.464,A -85,B 0,C 180,E1 3607.888,E2 3607.888} C_VEL
LIN {X 0,Y 202.141,Z 941.205,A -85,B 0,C 180,E1 3606.163,E2 3606.163} C_VEL
LIN {X 0,Y 203.49,Z 939.975,A -85,B 0,C 180,E1 3606.02,E2 3606.02} C_VEL
LIN {X 0,Y 186.612,Z 955.614,A -85,B 0,C 180,E1 3604.735,E2 3604.735} C_VEL
LIN {X 0,Y 168.202,Z 970.467,A -85,B 0,C 180,E1 3602.96,E2 3602.96} C_VEL
LIN {X 0,Y 147.984,Z 984.645,A -85,B 0,C 180,E1 3600.411,E2 3600.411} C_VEL
LIN {X 0,Y 128.161,Z 996.759,A -85,B 0,C 180,E1 3596.979,E2 3596.979} C_VEL
LIN {X 0,Y 119.644,Z 1001.416,A -85,B 0,C 180,E1 3595.107,E2 3595.107} C_VEL
LIN {X 0,Y 112.979,Z 1004.696,A -85,B 0,C 180,E1 3593.989,E2 3593.989} C_VEL
LIN {X 0,Y 93.437,Z 1012.298,A -85,B 0,C 180,E1 3592.02,E2 3592.02} C_VEL
LIN {X 0,Y 87.677,Z 1014.469,A -85,B 0,C 180,E1 3590.432,E2 3590.432} C_VEL
LIN {X 0,Y 68.878,Z 1021.748,A -85,B 0,C 180,E1 3580.499,E2 3580.499} C_VEL
LIN {X 0,Y 53.178,Z 1027.287,A -85,B 0,C 180,E1 3563.949,E2 3563.949} C_VEL
LIN {X 0,Y 44.454,Z 1030.889,A -85,B 0,C 180,E1 3539.658,E2 3539.658} C_VEL
LIN {X 0,Y 43.973,Z 1032.549,A -85,B 0,C 180,E1 3516.528,E2 3516.528} C_VEL
LIN {X 0,Y 44.802,Z 1032.848,A -85,B 0,C 180,E1 3510,E2 3510} C_VEL
LIN {X 0,Y 43.593,Z 1031.621,A -85,B 0,C 180,E1 3488.47,E2 3488.47} C_VEL
LIN {X 0,Y 49.158,Z 1028.722,A -85,B 0,C 180,E1 3463.748,E2 3463.748} C_VEL
LIN {X 0,Y 63.416,Z 1023.608,A -85,B 0,C 180,E1 3443.868,E2 3443.868} C_VEL
LIN {X 0,Y 80.905,Z 1017.183,A -85,B 0,C 180,E1 3432.491,E2 3432.491} C_VEL
LIN {X 0,Y 101.37,Z 1008.481,A -85,B 0,C 180,E1 3424.985,E2 3424.985} C_VEL
LIN {X 0,Y 121.985,Z 998.337,A -85,B 0,C 180,E1 3420.241,E2 3420.241} C_VEL
LIN {X 0,Y 142.17,Z 986.86,A -85,B 0,C 180,E1 3417.045,E2 3417.045} C_VEL
LIN {X 0,Y 161.639,Z 974.05,A -85,B 0,C 180,E1 3414.818,E2 3414.818} C_VEL
LIN {X 0,Y 175.601,Z 963.636,A -85,B 0,C 180,E1 3413.515,E2 3413.515} C_VEL
LIN {X 0,Y 157.762,Z 975.63,A -85,B 0,C 180,E1 3411.378,E2 3411.378} C_VEL
LIN {X 0,Y 138.762,Z 986.524,A -85,B 0,C 180,E1 3408.513,E2 3408.513} C_VEL
LIN {X 0,Y 120.167,Z 995.51,A -85,B 0,C 180,E1 3404.84,E2 3404.84} C_VEL
LIN {X 0,Y 101.294,Z 1002.967,A -85,B 0,C 180,E1 3399.676,E2 3399.676} C_VEL
LIN {X 0,Y 82.662,Z 1008.976,A -85,B 0,C 180,E1 3392.006,E2 3392.006} C_VEL
LIN {X 0,Y 66.076,Z 1013.268,A -85,B 0,C 180,E1 3380.511,E2 3380.511} C_VEL
LIN {X 0,Y 53.198,Z 1015.859,A -85,B 0,C 180,E1 3363.029,E2 3363.029} C_VEL
LIN {X 0,Y 46.71,Z 1016.939,A -85,B 0,C 180,E1 3339.861,E2 3339.861} C_VEL
LIN {X 0,Y 46.847,Z 1016.93,A -85,B 0,C 180,E1 3318.925,E2 3318.925} C_VEL
LIN {X 0,Y 54.12,Z 1015.702,A -85,B 0,C 180,E1 3295.06,E2 3295.06} C_VEL
LIN {X 0,Y 67.427,Z 1013.029,A -85,B 0,C 180,E1 3278.193,E2 3278.193} C_VEL
LIN {X 0,Y 84.246,Z 1008.606,A -85,B 0,C 180,E1 3267.11,E2 3267.11} C_VEL
LIN {X 0,Y 103.013,Z 1002.438,A -85,B 0,C 180,E1 3259.694,E2 3259.694} C_VEL
LIN {X 0,Y 121.963,Z 994.805,A -85,B 0,C 180,E1 3254.675,E2 3254.675} C_VEL
LIN {X 0,Y 141.015,Z 985.513,A -85,B 0,C 180,E1 3251.038,E2 3251.038} C_VEL
LIN {X 0,Y 159.651,Z 974.63,A -85,B 0,C 180,E1 3248.299,E2 3248.299} C_VEL
LIN {X 0,Y 175.394,Z 964.017,A -85,B 0,C 180,E1 3246.417,E2 3246.417} C_VEL
LIN {X 0,Y 156.494,Z 977.737,A -85,B 0,C 180,E1 3244.647,E2 3244.647} C_VEL
LIN {X 0,Y 136.072,Z 990.617,A -85,B 0,C 180,E1 3242.086,E2 3242.086} C_VEL
LIN {X 0,Y 115.718,Z 1001.737,A -85,B 0,C 180,E1 3238.516,E2 3238.516} C_VEL
LIN {X 0,Y 95.644,Z 1011.114,A -85,B 0,C 180,E1 3233.283,E2 3233.283} C_VEL
LIN {X 0,Y 87.677,Z 1014.469,A -85,B 0,C 180,E1 3230.432,E2 3230.432} C_VEL
LIN {X 0,Y 80.955,Z 1016.96,A -85,B 0,C 180,E1 3228.359,E2 3228.359} C_VEL
LIN {X 0,Y 61.33,Z 1022.218,A -85,B 0,C 180,E1 3223.294,E2 3223.294} C_VEL
LIN {X 0,Y 55.855,Z 1023.672,A -85,B 0,C 180,E1 3219.845,E2 3219.845} C_VEL
LIN {X 0,Y 41.22,Z 1028.092,A -85,B 0,C 180,E1 3198.76,E2 3198.76} C_VEL
LIN {X 0,Y 35.537,Z 1030.773,A -85,B 0,C 180,E1 3166.341,E2 3166.341} C_VEL
LIN {X 0,Y 36.748,Z 1031.453,A -85,B 0,C 180,E1 3150,E2 3150} C_VEL
LIN {X 0,Y 36.177,Z 1030.059,A -85,B 0,C 180,E1 3121.975,E2 3121.975} C_VEL
LIN {X 0,Y 44.043,Z 1027.176,A -85,B 0,C 180,E1 3095.186,E2 3095.186} C_VEL
LIN {X 0,Y 60.762,Z 1022.036,A -85,B 0,C 180,E1 3076.242,E2 3076.242} C_VEL
LIN {X 0,Y 80.443,Z 1015.323,A -85,B 0,C 180,E1 3066.087,E2 3066.087} C_VEL
LIN {X 0,Y 101.535,Z 1006.758,A -85,B 0,C 180,E1 3059.998,E2 3059.998} C_VEL
LIN {X 0,Y 122.252,Z 996.838,A -85,B 0,C 180,E1 3056.207,E2 3056.207} C_VEL
LIN {X 0,Y 143.137,Z 985.18,A -85,B 0,C 180,E1 3053.582,E2 3053.582} C_VEL
LIN {X 0,Y 147.421,Z 982.522,A -85,B 0,C 180,E1 3053.108,E2 3053.108} C_VEL
LIN {X 0,Y 127.827,Z 992.631,A -85,B 0,C 180,E1 3050.258,E2 3050.258} C_VEL
LIN {X 0,Y 108.04,Z 1001.027,A -85,B 0,C 180,E1 3046.345,E2 3046.345} C_VEL
LIN {X 0,Y 88.885,Z 1007.575,A -85,B 0,C 180,E1 3040.895,E2 3040.895} C_VEL
LIN {X 0,Y 69.206,Z 1012.88,A -85,B 0,C 180,E1 3031.8,E2 3031.8} C_VEL
LIN {X 0,Y 52.803,Z 1016.279,A -85,B 0,C 180,E1 3017.604,E2 3017.604} C_VEL
LIN {X 0,Y 41.694,Z 1017.944,A -85,B 0,C 180,E1 2995.573,E2 2995.573} C_VEL
LIN {X 0,Y 38.323,Z 1018.424,A -85,B 0,C 180,E1 2967.009,E2 2967.009} C_VEL
LIN {X 0,Y 42.864,Z 1017.8,A -85,B 0,C 180,E1 2940.669,E2 2940.669} C_VEL
LIN {X 0,Y 56.177,Z 1015.656,A -85,B 0,C 180,E1 2918.451,E2 2918.451} C_VEL
LIN {X 0,Y 73.294,Z 1012.02,A -85,B 0,C 180,E1 2905.795,E2 2905.795} C_VEL
LIN {X 0,Y 92.435,Z 1006.576,A -85,B 0,C 180,E1 2897.845,E2 2897.845} C_VEL
LIN {X 0,Y 111.735,Z 999.666,A -85,B 0,C 180,E1 2892.736,E2 2892.736} C_VEL
LIN {X 0,Y 130.665,Z 991.438,A -85,B 0,C 180,E1 2889.204,E2 2889.204} C_VEL
LIN {X 0,Y 147.243,Z 982.788,A -85,B 0,C 180,E1 2886.824,E2 2886.824} C_VEL
LIN {X 0,Y 126.352,Z 994.83,A -85,B 0,C 180,E1 2884.38,E2 2884.38} C_VEL
LIN {X 0,Y 104.995,Z 1005.339,A -85,B 0,C 180,E1 2880.743,E2 2880.743} C_VEL
LIN {X 0,Y 83.714,Z 1014.119,A -85,B 0,C 180,E1 2875.075,E2 2875.075} C_VEL
LIN {X 0,Y 62.997,Z 1021.373,A -85,B 0,C 180,E1 2865.292,E2 2865.292} C_VEL
LIN {X 0,Y 55.855,Z 1023.672,A -85,B 0,C 180,E1 2859.845,E2 2859.845} C_VEL
LIN {X 0,Y 49.673,Z 1025.186,A -85,B 0,C 180,E1 2854.988,E2 2854.988} C_VEL
LIN {X 0,Y 37.891,Z 1027.123,A -85,B 0,C 180,E1 2845.305,E2 2845.305} C_VEL
LIN {X 0,Y 30.886,Z 1028.168,A -85,B 0,C 180,E1 2833.295,E2 2833.295} C_VEL
LIN {X 0,Y 29.221,Z 1028.577,A -85,B 0,C 180,E1 2826.613,E2 2826.613} C_VEL
LIN {X 0,Y 28.659,Z 1030.052,A -85,B 0,C 180,E1 2790,E2 2790} C_VEL
LIN {X 0,Y 29.416,Z 1028.487,A -85,B 0,C 180,E1 2752.278,E2 2752.278} C_VEL
LIN {X 0,Y 41.709,Z 1025.263,A -85,B 0,C 180,E1 2722.549,E2 2722.549} C_VEL
LIN {X 0,Y 60.498,Z 1020.101,A -85,B 0,C 180,E1 2707.411,E2 2707.411} C_VEL
LIN {X 0,Y 82.999,Z 1012.713,A -85,B 0,C 180,E1 2699.138,E2 2699.138} C_VEL
LIN {X 0,Y 104.427,Z 1004.209,A -85,B 0,C 180,E1 2694.736,E2 2694.736} C_VEL
LIN {X 0,Y 118.96,Z 997.432,A -85,B 0,C 180,E1 2692.658,E2 2692.658} C_VEL
LIN {X 0,Y 98.715,Z 1005.119,A -85,B 0,C 180,E1 2688.903,E2 2688.903} C_VEL
LIN {X 0,Y 77.417,Z 1011.502,A -85,B 0,C 180,E1 2682.889,E2 2682.889} C_VEL
LIN {X 0,Y 58.149,Z 1015.873,A -85,B 0,C 180,E1 2673.398,E2 2673.398} C_VEL
LIN {X 0,Y 41.5,Z 1018.503,A -85,B 0,C 180,E1 2656.286,E2 2656.286} C_VEL
LIN {X 0,Y 31.286,Z 1019.671,A -85,B 0,C 180,E1 2624.814,E2 2624.814} C_VEL
LIN {X 0,Y 31.512,Z 1019.662,A -85,B 0,C 180,E1 2593.407,E2 2593.407} C_VEL
LIN {X 0,Y 42.133,Z 1018.444,A -85,B 0,C 180,E1 2562.637,E2 2562.637} C_VEL
LIN {X 0,Y 58.956,Z 1015.776,A -85,B 0,C 180,E1 2545.993,E2 2545.993} C_VEL
LIN {X 0,Y 78.3,Z 1011.355,A -85,B 0,C 180,E1 2536.72,E2 2536.72} C_VEL
LIN {X 0,Y 98.803,Z 1005.193,A -85,B 0,C 180,E1 2531.003,E2 2531.003} C_VEL
LIN {X 0,Y 118.693,Z 997.693,A -85,B 0,C 180,E1 2527.261,E2 2527.261} C_VEL
LIN {X 0,Y 97.225,Z 1007.286,A -85,B 0,C 180,E1 2524.009,E2 2524.009} C_VEL
LIN {X 0,Y 74.026,Z 1015.905,A -85,B 0,C 180,E1 2518.208,E2 2518.208} C_VEL
LIN {X 0,Y 53.122,Z 1022.3,A -85,B 0,C 180,E1 2508.168,E2 2508.168} C_VEL
LIN {X 0,Y 36.22,Z 1026.63,A -85,B 0,C 180,E1 2488.843,E2 2488.843} C_VEL
LIN {X 0,Y 29.221,Z 1028.577,A -85,B 0,C 180,E1 2466.613,E2 2466.613} C_VEL
LIN {X 0,Y 27.077,Z 1028.99,A -85,B 0,C 180,E1 2457.075,E2 2457.075} C_VEL
LIN {X 0,Y 23.62,Z 1028.964,A -85,B 0,C 180,E1 2443.952,E2 2443.952} C_VEL
LIN {X 0,Y 19.74,Z 1028.203,A -85,B 0,C 180,E1 2411.976,E2 2411.976} C_VEL
LIN {X 0,Y 28.894,Z 1025.964,A -85,B 0,C 180,E1 2364.528,E2 2364.528} C_VEL
LIN {X 0,Y 48.152,Z 1021.697,A -85,B 0,C 180,E1 2344.644,E2 2344.644} C_VEL
LIN {X 0,Y 71.173,Z 1015.332,A -85,B 0,C 180,E1 2335.899,E2 2335.899} C_VEL
LIN {X 0,Y 89.971,Z 1008.911,A -85,B 0,C 180,E1 2332.08,E2 2332.08} C_VEL
LIN {X 0,Y 68.864,Z 1014.467,A -85,B 0,C 180,E1 2326.607,E2 2326.607} C_VEL
LIN {X 0,Y 48.848,Z 1018.213,A -85,B 0,C 180,E1 2317.088,E2 2317.088} C_VEL
LIN {X 0,Y 30.77,Z 1020.461,A -85,B 0,C 180,E1 2295.635,E2 2295.635} C_VEL
LIN {X 0,Y 22.69,Z 1021.128,A -85,B 0,C 180,E1 2257.597,E2 2257.597} C_VEL
LIN {X 0,Y 27.695,Z 1020.758,A -85,B 0,C 180,E1 2212.14,E2 2212.14} C_VEL
LIN {X 0,Y 42.859,Z 1019.153,A -85,B 0,C 180,E1 2187.562,E2 2187.562} C_VEL
LIN {X 0,Y 62.331,Z 1015.877,A -85,B 0,C 180,E1 2175.747,E2 2175.747} C_VEL
LIN {X 0,Y 84.047,Z 1010.699,A -85,B 0,C 180,E1 2169.101,E2 2169.101} C_VEL
LIN {X 0,Y 89.825,Z 1009.054,A -85,B 0,C 180,E1 2167.829,E2 2167.829} C_VEL
LIN {X 0,Y 67.084,Z 1016.686,A -85,B 0,C 180,E1 2163.01,E2 2163.01} C_VEL
LIN {X 0,Y 45.276,Z 1022.417,A -85,B 0,C 180,E1 2153.599,E2 2153.599} C_VEL
LIN {X 0,Y 26.509,Z 1026.415,A -85,B 0,C 180,E1 2130.171,E2 2130.171} C_VEL
LIN {X 0,Y 19.745,Z 1028.291,A -85,B 0,C 180,E1 2084.666,E2 2084.666} C_VEL
LIN {X 0,Y 20.505,Z 1028.64,A -85,B 0,C 180,E1 2070,E2 2070} C_VEL
LIN {X 0,Y 19.74,Z 1028.203,A -85,B 0,C 180,E1 2051.976,E2 2051.976} C_VEL
LIN {X 0,Y 20.318,Z 1027.476,A -85,B 0,C 180,E1 2029.836,E2 2029.836} C_VEL
LIN {X 0,Y 31.056,Z 1023.801,A -85,B 0,C 180,E1 1984.514,E2 1984.514} C_VEL
LIN {X 0,Y 35.896,Z 1022.797,A -85,B 0,C 180,E1 1980.014,E2 1980.014} C_VEL
LIN {X 0,Y 58.619,Z 1017.689,A -85,B 0,C 180,E1 1971.617,E2 1971.617} C_VEL
LIN {X 0,Y 60.121,Z 1017.292,A -85,B 0,C 180,E1 1971.28,E2 1971.28} C_VEL
LIN {X 0,Y 38.916,Z 1020.58,A -85,B 0,C 180,E1 1961.924,E2 1961.924} C_VEL
LIN {X 0,Y 21.916,Z 1022.112,A -85,B 0,C 180,E1 1940.293,E2 1940.293} C_VEL
LIN {X 0,Y 14.907,Z 1022.5,A -85,B 0,C 180,E1 1878.392,E2 1878.392} C_VEL
LIN {X 0,Y 25.854,Z 1021.851,A -85,B 0,C 180,E1 1831.699,E2 1831.699} C_VEL
LIN {X 0,Y 46.568,Z 1019.602,A -85,B 0,C 180,E1 1813.665,E2 1813.665} C_VEL
LIN {X 0,Y 59.836,Z 1017.419,A -85,B 0,C 180,E1 1808.653,E2 1808.653} C_VEL
LIN {X 0,Y 36.997,Z 1022.626,A -85,B 0,C 180,E1 1800.64,E2 1800.64} C_VEL
LIN {X 0,Y 17.555,Z 1025.865,A -85,B 0,C 180,E1 1775.685,E2 1775.685} C_VEL
LIN {X 0,Y 12.318,Z 1027.221,A -85,B 0,C 180,E1 1709.999,E2 1709.999} C_VEL
LIN {X 0,Y 20.466,Z 1025.39,A -85,B 0,C 180,E1 1637.036,E2 1637.036} C_VEL
LIN {X 0,Y 35.896,Z 1022.797,A -85,B 0,C 180,E1 1620.014,E2 1620.014} C_VEL
LIN {X 0,Y 34.425,Z 1022.849,A -85,B 0,C 180,E1 1618.588,E2 1618.588} C_VEL
LIN {X 0,Y 26.625,Z 1023.705,A -85,B 0,C 180,E1 1618.129,E2 1618.129} C_VEL
LIN {X 0,Y 8.838,Z 1025.257,A -85,B 0,C 180,E1 1632.516,E2 1632.516} C_VEL
LIN {X 0,Y 3.97,Z 1025.757,A -85,B 0,C 180,E1 1701.231,E2 1701.231} C_VEL
LIN {X 0,Y 3.935,Z 1025.734,A -85,B 0,C 180,E1 1724.717,E2 1724.717} C_VEL
LIN {X 0,Y 20.163,Z 1023.892,A -85,B 0,C 180,E1 1807.36,E2 1807.36} C_VEL
LIN {X 0,Y 27.497,Z 1022.937,A -85,B 0,C 180,E1 1810.949,E2 1810.949} C_VEL
LIN {X 0,Y 9.627,Z 1023.793,A -85,B 0,C 180,E1 1843.363,E2 1843.363} C_VEL
LIN {X 0,Y 11.928,Z 1023.737,A -85,B 0,C 180,E1 1946.954,E2 1946.954} C_VEL
LIN {X 0,Y 27.483,Z 1022.922,A -85,B 0,C 180,E1 1969.205,E2 1969.205} C_VEL
LIN {X 0,Y 7.044,Z 1025.283,A -85,B 0,C 180,E1 1996.466,E2 1996.466} C_VEL
LIN {X 0,Y 3.97,Z 1025.757,A -85,B 0,C 180,E1 2061.231,E2 2061.231} C_VEL
LIN {X 0,Y 4.606,Z 1027.752,A -85,B 0,C 180,E1 2084.799,E2 2084.799} C_VEL
LIN {X 0,Y 4.606,Z 1104,A -85,B 0,C 180,E1 2084.799,E2 2084.799} C_VEL
LIN {X 0,Y 4.606,Z 1104,A -85,B 0,C 180,E1 2084.799,E2 2084.799}

QRS_NEXT_CUT()

QRS_NEXT()
QRS_HOME()

END
